LIN {X 0,Y 334.307,Z 627.426,A -85,B 0,C 180,E1 -14365.347,E2 -14365.347} C_VEL
LIN {X 0,Y 334.182,Z 628.158,A -85,B 0,C 180,E1 -14365.662,E2 -14365.662} C_VEL
LIN {X 0,Y 334.072,Z 630.189,A -85,B 0,C 180,E1 -14366.548,E2 -14366.548} C_VEL
LIN {X 0,Y 336.803,Z 644.466,A -85,B 0,C 180,E1 -14367.297,E2 -14367.297} C_VEL
LIN {X 0,Y 339.056,Z 657.276,A -85,B 0,C 180,E1 -14368.193,E2 -14368.193} C_VEL
LIN {X 0,Y 338.208,Z 670.123,A -85,B 0,C 180,E1 -14369.223,E2 -14369.223} C_VEL
LIN {X 0,Y 337.091,Z 682.489,A -85,B 0,C 180,E1 -14370.492,E2 -14370.492} C_VEL
LIN {X 0,Y 336.021,Z 693.493,A -85,B 0,C 180,E1 -14371.928,E2 -14371.928} C_VEL
LIN {X 0,Y 335.044,Z 703.461,A -85,B 0,C 180,E1 -14373.529,E2 -14373.529} C_VEL
LIN {X 0,Y 334.192,Z 711.545,A -85,B 0,C 180,E1 -14375.128,E2 -14375.128} C_VEL
LIN {X 0,Y 333.445,Z 719.422,A -85,B 0,C 180,E1 -14377.051,E2 -14377.051} C_VEL
LIN {X 0,Y 332.869,Z 725.659,A -85,B 0,C 180,E1 -14378.966,E2 -14378.966} C_VEL
LIN {X 0,Y 332.483,Z 730.459,A -85,B 0,C 180,E1 -14380.875,E2 -14380.875} C_VEL
LIN {X 0,Y 332.219,Z 734.042,A -85,B 0,C 180,E1 -14382.773,E2 -14382.773} C_VEL
LIN {X 0,Y 332.056,Z 735.815,A -85,B 0,C 180,E1 -14384.03,E2 -14384.03} C_VEL
LIN {X 0,Y 332.023,Z 737.142,A -85,B 0,C 180,E1 -14385.286,E2 -14385.286} C_VEL
LIN {X 0,Y 332.085,Z 738.091,A -85,B 0,C 180,E1 -14386.776,E2 -14386.776} C_VEL
LIN {X 0,Y 332.139,Z 738.414,A -85,B 0,C 180,E1 -14389.022,E2 -14389.022} C_VEL
LIN {X 0,Y 332.284,Z 737.954,A -85,B 0,C 180,E1 -14390.259,E2 -14390.259} C_VEL
LIN {X 0,Y 332.509,Z 737.089,A -85,B 0,C 180,E1 -14391.492,E2 -14391.492} C_VEL
LIN {X 0,Y 332.844,Z 735.56,A -85,B 0,C 180,E1 -14392.92,E2 -14392.92} C_VEL
LIN {X 0,Y 333.43,Z 731.936,A -85,B 0,C 180,E1 -14395.164,E2 -14395.164} C_VEL
LIN {X 0,Y 334.131,Z 727.836,A -85,B 0,C 180,E1 -14396.986,E2 -14396.986} C_VEL
LIN {X 0,Y 335.257,Z 721.578,A -85,B 0,C 180,E1 -14399.1,E2 -14399.1} C_VEL
LIN {X 0,Y 336.526,Z 714.727,A -85,B 0,C 180,E1 -14400.898,E2 -14400.898} C_VEL
LIN {X 0,Y 337.99,Z 706.462,A -85,B 0,C 180,E1 -14402.651,E2 -14402.651} C_VEL
LIN {X 0,Y 339.489,Z 697.76,A -85,B 0,C 180,E1 -14404.156,E2 -14404.156} C_VEL
LIN {X 0,Y 341.171,Z 687.321,A -85,B 0,C 180,E1 -14405.616,E2 -14405.616} C_VEL
LIN {X 0,Y 342.749,Z 675.77,A -85,B 0,C 180,E1 -14406.919,E2 -14406.919} C_VEL
LIN {X 0,Y 344.181,Z 663.857,A -85,B 0,C 180,E1 -14407.968,E2 -14407.968} C_VEL
LIN {X 0,Y 342.351,Z 652.946,A -85,B 0,C 180,E1 -14409.036,E2 -14409.036} C_VEL
LIN {X 0,Y 338.669,Z 640.492,A -85,B 0,C 180,E1 -14410.207,E2 -14410.207} C_VEL
LIN {X 0,Y 336.47,Z 634.41,A -85,B 0,C 180,E1 -14410.786,E2 -14410.786} C_VEL
LIN {X 0,Y 337.122,Z 626.531,A -85,B 0,C 180,E1 -14414.488,E2 -14414.488} C_VEL
LIN {X 0,Y 337.867,Z 618.773,A -85,B 0,C 180,E1 -14418.181,E2 -14418.181} C_VEL
LIN {X 0,Y 338.839,Z 611.142,A -85,B 0,C 180,E1 -14421.923,E2 -14421.923} C_VEL
LIN {X 0,Y 339.229,Z 606.089,A -85,B 0,C 180,E1 -14424.479,E2 -14424.479} C_VEL
LIN {X 0,Y 338.754,Z 601.9,A -85,B 0,C 180,E1 -14426.865,E2 -14426.865} C_VEL
LIN {X 0,Y 337.834,Z 597.015,A -85,B 0,C 180,E1 -14429.953,E2 -14429.953} C_VEL
LIN {X 0,Y 336.765,Z 592.554,A -85,B 0,C 180,E1 -14433.411,E2 -14433.411} C_VEL
LIN {X 0,Y 335.981,Z 589.986,A -85,B 0,C 180,E1 -14435.853,E2 -14435.853} C_VEL
LIN {X 0,Y 335.211,Z 587.549,A -85,B 0,C 180,E1 -14438.975,E2 -14438.975} C_VEL
LIN {X 0,Y 334.904,Z 586.539,A -85,B 0,C 180,E1 -14440.936,E2 -14440.936} C_VEL
LIN {X 0,Y 334.499,Z 586.598,A -85,B 0,C 180,E1 -14441.944,E2 -14441.944} C_VEL
LIN {X 0,Y 335.969,Z 593.434,A -85,B 0,C 180,E1 -14445.336,E2 -14445.336} C_VEL
LIN {X 0,Y 337.645,Z 601.963,A -85,B 0,C 180,E1 -14449.226,E2 -14449.226} C_VEL
LIN {X 0,Y 338.527,Z 607.233,A -85,B 0,C 180,E1 -14451.48,E2 -14451.48} C_VEL
LIN {X 0,Y 338.397,Z 611.019,A -85,B 0,C 180,E1 -14452.968,E2 -14452.968} C_VEL
LIN {X 0,Y 336.894,Z 620.66,A -85,B 0,C 180,E1 -14456.559,E2 -14456.559} C_VEL
LIN {X 0,Y 335.74,Z 629.739,A -85,B 0,C 180,E1 -14459.843,E2 -14459.843} C_VEL
LIN {X 0,Y 334.739,Z 639.124,A -85,B 0,C 180,E1 -14463.168,E2 -14463.168} C_VEL
LIN {X 0,Y 334.472,Z 641.914,A -85,B 0,C 180,E1 -14464.13,E2 -14464.13} C_VEL
LIN {X 0,Y 335.666,Z 653.856,A -85,B 0,C 180,E1 -14465.905,E2 -14465.905} C_VEL
LIN {X 0,Y 336.107,Z 656.378,A -85,B 0,C 180,E1 -14466.191,E2 -14466.191} C_VEL
LIN {X 0,Y 339.515,Z 671.747,A -85,B 0,C 180,E1 -14467.228,E2 -14467.228} C_VEL
LIN {X 0,Y 340.677,Z 682.969,A -85,B 0,C 180,E1 -14467.991,E2 -14467.991} C_VEL
LIN {X 0,Y 340.835,Z 696.04,A -85,B 0,C 180,E1 -14468.978,E2 -14468.978} C_VEL
LIN {X 0,Y 340.476,Z 708.153,A -85,B 0,C 180,E1 -14470.089,E2 -14470.089} C_VEL
LIN {X 0,Y 339.636,Z 716.55,A -85,B 0,C 180,E1 -14470.981,E2 -14470.981} C_VEL
LIN {X 0,Y 337.998,Z 727.237,A -85,B 0,C 180,E1 -14472.297,E2 -14472.297} C_VEL
LIN {X 0,Y 336.398,Z 737.43,A -85,B 0,C 180,E1 -14473.845,E2 -14473.845} C_VEL
LIN {X 0,Y 335.114,Z 745.944,A -85,B 0,C 180,E1 -14475.425,E2 -14475.425} C_VEL
LIN {X 0,Y 334.012,Z 753.925,A -85,B 0,C 180,E1 -14477.237,E2 -14477.237} C_VEL
LIN {X 0,Y 333.133,Z 760.378,A -85,B 0,C 180,E1 -14479.056,E2 -14479.056} C_VEL
LIN {X 0,Y 332.615,Z 765.591,A -85,B 0,C 180,E1 -14480.883,E2 -14480.883} C_VEL
LIN {X 0,Y 332.292,Z 769.66,A -85,B 0,C 180,E1 -14482.711,E2 -14482.711} C_VEL
LIN {X 0,Y 332.201,Z 771.787,A -85,B 0,C 180,E1 -14483.929,E2 -14483.929} C_VEL
LIN {X 0,Y 332.179,Z 773.487,A -85,B 0,C 180,E1 -14485.146,E2 -14485.146} C_VEL
LIN {X 0,Y 332.155,Z 774.712,A -85,B 0,C 180,E1 -14486.362,E2 -14486.362} C_VEL
LIN {X 0,Y 332.2,Z 775.52,A -85,B 0,C 180,E1 -14487.576,E2 -14487.576} C_VEL
LIN {X 0,Y 332.339,Z 775.927,A -85,B 0,C 180,E1 -14488.789,E2 -14488.789} C_VEL
LIN {X 0,Y 332.37,Z 775.897,A -85,B 0,C 180,E1 -14490.001,E2 -14490.001} C_VEL
LIN {X 0,Y 332.374,Z 775.4,A -85,B 0,C 180,E1 -14491.213,E2 -14491.213} C_VEL
LIN {X 0,Y 332.287,Z 774.481,A -85,B 0,C 180,E1 -14492.425,E2 -14492.425} C_VEL
LIN {X 0,Y 332.186,Z 773.133,A -85,B 0,C 180,E1 -14493.64,E2 -14493.64} C_VEL
LIN {X 0,Y 332.298,Z 771.3,A -85,B 0,C 180,E1 -14494.854,E2 -14494.854} C_VEL
LIN {X 0,Y 332.272,Z 767.789,A -85,B 0,C 180,E1 -14496.621,E2 -14496.621} C_VEL
LIN {X 0,Y 332.466,Z 762.816,A -85,B 0,C 180,E1 -14498.511,E2 -14498.511} C_VEL
LIN {X 0,Y 332.84,Z 756.668,A -85,B 0,C 180,E1 -14500.34,E2 -14500.34} C_VEL
LIN {X 0,Y 333.491,Z 748.981,A -85,B 0,C 180,E1 -14502.167,E2 -14502.167} C_VEL
LIN {X 0,Y 334.174,Z 741.078,A -85,B 0,C 180,E1 -14503.687,E2 -14503.687} C_VEL
LIN {X 0,Y 334.972,Z 732.11,A -85,B 0,C 180,E1 -14505.111,E2 -14505.111} C_VEL
LIN {X 0,Y 336.113,Z 720.935,A -85,B 0,C 180,E1 -14506.554,E2 -14506.554} C_VEL
LIN {X 0,Y 337.216,Z 709.113,A -85,B 0,C 180,E1 -14507.747,E2 -14507.747} C_VEL
LIN {X 0,Y 336.932,Z 696.74,A -85,B 0,C 180,E1 -14508.767,E2 -14508.767} C_VEL
LIN {X 0,Y 336.181,Z 683.119,A -85,B 0,C 180,E1 -14509.613,E2 -14509.613} C_VEL
LIN {X 0,Y 335.029,Z 669.463,A -85,B 0,C 180,E1 -14510.221,E2 -14510.221} C_VEL
LIN {X 0,Y 333.69,Z 657.114,A -85,B 0,C 180,E1 -14510.739,E2 -14510.739} C_VEL
LIN {X 0,Y 333.319,Z 651.132,A -85,B 0,C 180,E1 -14511.242,E2 -14511.242} C_VEL
LIN {X 0,Y 334.083,Z 638.01,A -85,B 0,C 180,E1 -14515.644,E2 -14515.644} C_VEL
LIN {X 0,Y 335.042,Z 626.598,A -85,B 0,C 180,E1 -14519.535,E2 -14519.535} C_VEL
LIN {X 0,Y 336.106,Z 615.846,A -85,B 0,C 180,E1 -14523.237,E2 -14523.237} C_VEL
LIN {X 0,Y 337.236,Z 605.77,A -85,B 0,C 180,E1 -14526.81,E2 -14526.81} C_VEL
LIN {X 0,Y 337.323,Z 602.151,A -85,B 0,C 180,E1 -14528.132,E2 -14528.132} C_VEL
LIN {X 0,Y 335.692,Z 593.071,A -85,B 0,C 180,E1 -14531.692,E2 -14531.692} C_VEL
LIN {X 0,Y 334.038,Z 584.825,A -85,B 0,C 180,E1 -14535.121,E2 -14535.121} C_VEL
LIN {X 0,Y 333.645,Z 582.926,A -85,B 0,C 180,E1 -14535.962,E2 -14535.962} C_VEL
LIN {X 0,Y 333.652,Z 582.927,A -85,B 0,C 180,E1 -14539.315,E2 -14539.315} C_VEL
LIN {X 0,Y 333.672,Z 582.919,A -85,B 0,C 180,E1 -14543.167,E2 -14543.167} C_VEL
LIN {X 0,Y 333.644,Z 582.923,A -85,B 0,C 180,E1 -14546.792,E2 -14546.792} C_VEL
LIN {X 0,Y 333.709,Z 582.914,A -85,B 0,C 180,E1 -14549.71,E2 -14549.71} C_VEL
LIN {X 0,Y 333.74,Z 582.911,A -85,B 0,C 180,E1 -14553.754,E2 -14553.754} C_VEL
LIN {X 0,Y 333.725,Z 582.914,A -85,B 0,C 180,E1 -14557.914,E2 -14557.914} C_VEL
LIN {X 0,Y 333.799,Z 582.903,A -85,B 0,C 180,E1 -14561.589,E2 -14561.589} C_VEL
LIN {X 0,Y 333.813,Z 582.901,A -85,B 0,C 180,E1 -14565.576,E2 -14565.576} C_VEL
LIN {X 0,Y 333.838,Z 582.898,A -85,B 0,C 180,E1 -14569.078,E2 -14569.078} C_VEL
LIN {X 0,Y 334.031,Z 582.876,A -85,B 0,C 180,E1 -14572.747,E2 -14572.747} C_VEL
LIN {X 0,Y 333.813,Z 582.901,A -85,B 0,C 180,E1 -14575.169,E2 -14575.169} C_VEL
LIN {X 0,Y 334.109,Z 582.864,A -85,B 0,C 180,E1 -14577.588,E2 -14577.588} C_VEL
LIN {X 0,Y 334.252,Z 582.848,A -85,B 0,C 180,E1 -14580,E2 -14580} C_VEL
LIN {X 0,Y 334.109,Z 582.869,A -85,B 0,C 180,E1 -14582.411,E2 -14582.411} C_VEL
LIN {X 0,Y 334.029,Z 582.873,A -85,B 0,C 180,E1 -14587.252,E2 -14587.252} C_VEL
LIN {X 0,Y 333.837,Z 582.899,A -85,B 0,C 180,E1 -14590.921,E2 -14590.921} C_VEL
LIN {X 0,Y 333.812,Z 582.904,A -85,B 0,C 180,E1 -14594.634,E2 -14594.634} C_VEL
LIN {X 0,Y 333.8,Z 582.906,A -85,B 0,C 180,E1 -14598.655,E2 -14598.655} C_VEL
LIN {X 0,Y 333.695,Z 582.919,A -85,B 0,C 180,E1 -14602.277,E2 -14602.277} C_VEL
LIN {X 0,Y 333.739,Z 582.913,A -85,B 0,C 180,E1 -14606.245,E2 -14606.245} C_VEL
LIN {X 0,Y 333.713,Z 582.914,A -85,B 0,C 180,E1 -14608.971,E2 -14608.971} C_VEL
LIN {X 0,Y 333.645,Z 582.926,A -85,B 0,C 180,E1 -14612.586,E2 -14612.586} C_VEL
LIN {X 0,Y 333.678,Z 582.92,A -85,B 0,C 180,E1 -14616.138,E2 -14616.138} C_VEL
LIN {X 0,Y 333.649,Z 582.921,A -85,B 0,C 180,E1 -14619.191,E2 -14619.191} C_VEL
LIN {X 0,Y 333.636,Z 582.928,A -85,B 0,C 180,E1 -14622.499,E2 -14622.499} C_VEL
LIN {X 0,Y 333.621,Z 582.925,A -85,B 0,C 180,E1 -14625.958,E2 -14625.958} C_VEL
LIN {X 0,Y 333.648,Z 582.921,A -85,B 0,C 180,E1 -14629.314,E2 -14629.314} C_VEL
LIN {X 0,Y 333.667,Z 582.919,A -85,B 0,C 180,E1 -14633.166,E2 -14633.166} C_VEL
LIN {X 0,Y 333.637,Z 582.925,A -85,B 0,C 180,E1 -14636.791,E2 -14636.791} C_VEL
LIN {X 0,Y 333.695,Z 582.915,A -85,B 0,C 180,E1 -14639.712,E2 -14639.712} C_VEL
LIN {X 0,Y 333.74,Z 582.914,A -85,B 0,C 180,E1 -14642.4,E2 -14642.4} C_VEL
LIN {X 0,Y 333.727,Z 582.912,A -85,B 0,C 180,E1 -14645.09,E2 -14645.09} C_VEL
LIN {X 0,Y 333.685,Z 582.918,A -85,B 0,C 180,E1 -14649.019,E2 -14649.019} C_VEL
LIN {X 0,Y 333.793,Z 582.903,A -85,B 0,C 180,E1 -14651.588,E2 -14651.588} C_VEL
LIN {X 0,Y 333.808,Z 582.901,A -85,B 0,C 180,E1 -14655.575,E2 -14655.575} C_VEL
LIN {X 0,Y 333.837,Z 582.899,A -85,B 0,C 180,E1 -14659.077,E2 -14659.077} C_VEL
LIN {X 0,Y 334.025,Z 582.879,A -85,B 0,C 180,E1 -14662.746,E2 -14662.746} C_VEL
LIN {X 0,Y 333.936,Z 582.889,A -85,B 0,C 180,E1 -14664.375,E2 -14664.375} C_VEL
LIN {X 0,Y 337.247,Z 594.141,A -85,B 0,C 180,E1 -14665.357,E2 -14665.357} C_VEL
LIN {X 0,Y 339.912,Z 603.552,A -85,B 0,C 180,E1 -14666.339,E2 -14666.339} C_VEL
LIN {X 0,Y 339.161,Z 614.359,A -85,B 0,C 180,E1 -14667.487,E2 -14667.487} C_VEL
LIN {X 0,Y 338.331,Z 624.38,A -85,B 0,C 180,E1 -14668.809,E2 -14668.809} C_VEL
LIN {X 0,Y 337.349,Z 634.006,A -85,B 0,C 180,E1 -14670.388,E2 -14670.388} C_VEL
LIN {X 0,Y 336.455,Z 642.391,A -85,B 0,C 180,E1 -14672.094,E2 -14672.094} C_VEL
LIN {X 0,Y 335.7,Z 649.55,A -85,B 0,C 180,E1 -14673.9,E2 -14673.9} C_VEL
LIN {X 0,Y 335.16,Z 654.395,A -85,B 0,C 180,E1 -14675.413,E2 -14675.413} C_VEL
LIN {X 0,Y 334.655,Z 659.115,A -85,B 0,C 180,E1 -14677.238,E2 -14677.238} C_VEL
LIN {X 0,Y 334.241,Z 662.263,A -85,B 0,C 180,E1 -14678.793,E2 -14678.793} C_VEL
LIN {X 0,Y 333.988,Z 665.37,A -85,B 0,C 180,E1 -14680.916,E2 -14680.916} C_VEL
LIN {X 0,Y 333.91,Z 666.609,A -85,B 0,C 180,E1 -14682.149,E2 -14682.149} C_VEL
LIN {X 0,Y 333.934,Z 667.776,A -85,B 0,C 180,E1 -14684.509,E2 -14684.509} C_VEL
LIN {X 0,Y 334.096,Z 667.803,A -85,B 0,C 180,E1 -14685.869,E2 -14685.869} C_VEL
LIN {X 0,Y 334.249,Z 667.398,A -85,B 0,C 180,E1 -14687.118,E2 -14687.118} C_VEL
LIN {X 0,Y 334.756,Z 665.826,A -85,B 0,C 180,E1 -14689.137,E2 -14689.137} C_VEL
LIN {X 0,Y 335.561,Z 662.549,A -85,B 0,C 180,E1 -14691.5,E2 -14691.5} C_VEL
LIN {X 0,Y 336.414,Z 658.718,A -85,B 0,C 180,E1 -14693.385,E2 -14693.385} C_VEL
LIN {X 0,Y 337.428,Z 653.667,A -85,B 0,C 180,E1 -14695.274,E2 -14695.274} C_VEL
LIN {X 0,Y 338.646,Z 647.151,A -85,B 0,C 180,E1 -14697.165,E2 -14697.165} C_VEL
LIN {X 0,Y 340.117,Z 638.895,A -85,B 0,C 180,E1 -14699.05,E2 -14699.05} C_VEL
LIN {X 0,Y 341.533,Z 630.236,A -85,B 0,C 180,E1 -14700.633,E2 -14700.633} C_VEL
LIN {X 0,Y 342.769,Z 620.752,A -85,B 0,C 180,E1 -14702.04,E2 -14702.04} C_VEL
LIN {X 0,Y 343.821,Z 612.329,A -85,B 0,C 180,E1 -14703.064,E2 -14703.064} C_VEL
LIN {X 0,Y 343.026,Z 608.47,A -85,B 0,C 180,E1 -14703.584,E2 -14703.584} C_VEL
LIN {X 0,Y 339.681,Z 597.97,A -85,B 0,C 180,E1 -14704.932,E2 -14704.932} C_VEL
LIN {X 0,Y 335.979,Z 588.61,A -85,B 0,C 180,E1 -14706.014,E2 -14706.014} C_VEL
LIN {X 0,Y 334.161,Z 585.204,A -85,B 0,C 180,E1 -14706.423,E2 -14706.423} C_VEL
LIN {X 0,Y 335.344,Z 592.252,A -85,B 0,C 180,E1 -14709.73,E2 -14709.73} C_VEL
LIN {X 0,Y 335.556,Z 597.441,A -85,B 0,C 180,E1 -14712.082,E2 -14712.082} C_VEL
LIN {X 0,Y 335.238,Z 605.006,A -85,B 0,C 180,E1 -14715.46,E2 -14715.46} C_VEL
LIN {X 0,Y 334.771,Z 613.229,A -85,B 0,C 180,E1 -14719.09,E2 -14719.09} C_VEL
LIN {X 0,Y 334.502,Z 620.877,A -85,B 0,C 180,E1 -14722.462,E2 -14722.462} C_VEL
LIN {X 0,Y 334.182,Z 628.158,A -85,B 0,C 180,E1 -14725.662,E2 -14725.662} C_VEL
LIN {X 0,Y 334.028,Z 630.109,A -85,B 0,C 180,E1 -14726.142,E2 -14726.142} C_VEL
LIN {X 0,Y 333.66,Z 633.986,A -85,B 0,C 180,E1 -14726.58,E2 -14726.58} C_VEL
LIN {X 0,Y 333.01,Z 640.169,A -85,B 0,C 180,E1 -14726.906,E2 -14726.906} C_VEL
LIN {X 0,Y 331.643,Z 652.47,A -85,B 0,C 180,E1 -14727.534,E2 -14727.534} C_VEL
LIN {X 0,Y 331.953,Z 656.912,A -85,B 0,C 180,E1 -14727.855,E2 -14727.855} C_VEL
LIN {X 0,Y 331.934,Z 661.668,A -85,B 0,C 180,E1 -14728.218,E2 -14728.218} C_VEL
LIN {X 0,Y 331.085,Z 672.909,A -85,B 0,C 180,E1 -14729.196,E2 -14729.196} C_VEL
LIN {X 0,Y 329.945,Z 684.661,A -85,B 0,C 180,E1 -14730.491,E2 -14730.491} C_VEL
LIN {X 0,Y 328.887,Z 695.368,A -85,B 0,C 180,E1 -14731.959,E2 -14731.959} C_VEL
LIN {X 0,Y 327.925,Z 704.858,A -85,B 0,C 180,E1 -14733.568,E2 -14733.568} C_VEL
LIN {X 0,Y 326.893,Z 714.317,A -85,B 0,C 180,E1 -14735.553,E2 -14735.553} C_VEL
LIN {X 0,Y 326.186,Z 722.052,A -85,B 0,C 180,E1 -14737.63,E2 -14737.63} C_VEL
LIN {X 0,Y 325.593,Z 728.357,A -85,B 0,C 180,E1 -14739.797,E2 -14739.797} C_VEL
LIN {X 0,Y 325.274,Z 732.938,A -85,B 0,C 180,E1 -14741.925,E2 -14741.925} C_VEL
LIN {X 0,Y 325.009,Z 735.702,A -85,B 0,C 180,E1 -14743.674,E2 -14743.674} C_VEL
LIN {X 0,Y 324.943,Z 737.164,A -85,B 0,C 180,E1 -14744.958,E2 -14744.958} C_VEL
LIN {X 0,Y 324.993,Z 738.421,A -85,B 0,C 180,E1 -14746.68,E2 -14746.68} C_VEL
LIN {X 0,Y 325.05,Z 738.884,A -85,B 0,C 180,E1 -14748.78,E2 -14748.78} C_VEL
LIN {X 0,Y 325.179,Z 738.61,A -85,B 0,C 180,E1 -14750.044,E2 -14750.044} C_VEL
LIN {X 0,Y 325.389,Z 737.888,A -85,B 0,C 180,E1 -14751.305,E2 -14751.305} C_VEL
LIN {X 0,Y 325.784,Z 736.389,A -85,B 0,C 180,E1 -14752.89,E2 -14752.89} C_VEL
LIN {X 0,Y 326.358,Z 733.212,A -85,B 0,C 180,E1 -14755.059,E2 -14755.059} C_VEL
LIN {X 0,Y 327.053,Z 729.361,A -85,B 0,C 180,E1 -14756.921,E2 -14756.921} C_VEL
LIN {X 0,Y 328.051,Z 724.353,A -85,B 0,C 180,E1 -14758.773,E2 -14758.773} C_VEL
LIN {X 0,Y 329.521,Z 716.955,A -85,B 0,C 180,E1 -14760.917,E2 -14760.917} C_VEL
LIN {X 0,Y 331.111,Z 708.756,A -85,B 0,C 180,E1 -14762.778,E2 -14762.778} C_VEL
LIN {X 0,Y 332.902,Z 699.065,A -85,B 0,C 180,E1 -14764.541,E2 -14764.541} C_VEL
LIN {X 0,Y 334.651,Z 688.804,A -85,B 0,C 180,E1 -14766.028,E2 -14766.028} C_VEL
LIN {X 0,Y 336.327,Z 677.58,A -85,B 0,C 180,E1 -14767.354,E2 -14767.354} C_VEL
LIN {X 0,Y 337.802,Z 666.688,A -85,B 0,C 180,E1 -14768.375,E2 -14768.375} C_VEL
LIN {X 0,Y 337.714,Z 663.23,A -85,B 0,C 180,E1 -14768.709,E2 -14768.709} C_VEL
LIN {X 0,Y 336.082,Z 654.225,A -85,B 0,C 180,E1 -14769.631,E2 -14769.631} C_VEL
LIN {X 0,Y 332.251,Z 641.507,A -85,B 0,C 180,E1 -14770.925,E2 -14770.925} C_VEL
LIN {X 0,Y 329.847,Z 634.887,A -85,B 0,C 180,E1 -14771.616,E2 -14771.616} C_VEL
LIN {X 0,Y 330.567,Z 627.015,A -85,B 0,C 180,E1 -14775.412,E2 -14775.412} C_VEL
LIN {X 0,Y 331.423,Z 619.333,A -85,B 0,C 180,E1 -14779.189,E2 -14779.189} C_VEL
LIN {X 0,Y 332.525,Z 611.787,A -85,B 0,C 180,E1 -14783.017,E2 -14783.017} C_VEL
LIN {X 0,Y 332.695,Z 608.178,A -85,B 0,C 180,E1 -14784.992,E2 -14784.992} C_VEL
LIN {X 0,Y 332.133,Z 603.529,A -85,B 0,C 180,E1 -14787.745,E2 -14787.745} C_VEL
LIN {X 0,Y 331.628,Z 600.722,A -85,B 0,C 180,E1 -14789.673,E2 -14789.673} C_VEL
LIN {X 0,Y 331.003,Z 597.785,A -85,B 0,C 180,E1 -14792.061,E2 -14792.061} C_VEL
LIN {X 0,Y 330.159,Z 594.47,A -85,B 0,C 180,E1 -14795.082,E2 -14795.082} C_VEL
LIN {X 0,Y 329.451,Z 592.024,A -85,B 0,C 180,E1 -14798.218,E2 -14798.218} C_VEL
LIN {X 0,Y 329.268,Z 591.122,A -85,B 0,C 180,E1 -14799.817,E2 -14799.817} C_VEL
LIN {X 0,Y 328.816,Z 590.694,A -85,B 0,C 180,E1 -14801.578,E2 -14801.578} C_VEL
LIN {X 0,Y 328.227,Z 590.987,A -85,B 0,C 180,E1 -14803.171,E2 -14803.171} C_VEL
LIN {X 0,Y 329.616,Z 597.705,A -85,B 0,C 180,E1 -14806.465,E2 -14806.465} C_VEL
LIN {X 0,Y 331.329,Z 606.54,A -85,B 0,C 180,E1 -14810.482,E2 -14810.482} C_VEL
LIN {X 0,Y 331.645,Z 610.34,A -85,B 0,C 180,E1 -14812.083,E2 -14812.083} C_VEL
LIN {X 0,Y 330.527,Z 617.8,A -85,B 0,C 180,E1 -14814.965,E2 -14814.965} C_VEL
LIN {X 0,Y 328.965,Z 628.992,A -85,B 0,C 180,E1 -14819.155,E2 -14819.155} C_VEL
LIN {X 0,Y 327.834,Z 638.822,A -85,B 0,C 180,E1 -14822.685,E2 -14822.685} C_VEL
LIN {X 0,Y 329.077,Z 652.142,A -85,B 0,C 180,E1 -14824.885,E2 -14824.885} C_VEL
LIN {X 0,Y 329.478,Z 655.573,A -85,B 0,C 180,E1 -14825.358,E2 -14825.358} C_VEL
LIN {X 0,Y 332.741,Z 669.626,A -85,B 0,C 180,E1 -14826.398,E2 -14826.398} C_VEL
LIN {X 0,Y 334.185,Z 679.781,A -85,B 0,C 180,E1 -14827.127,E2 -14827.127} C_VEL
LIN {X 0,Y 334.605,Z 692.047,A -85,B 0,C 180,E1 -14828.062,E2 -14828.062} C_VEL
LIN {X 0,Y 334.086,Z 704.814,A -85,B 0,C 180,E1 -14829.209,E2 -14829.209} C_VEL
LIN {X 0,Y 333.568,Z 713.591,A -85,B 0,C 180,E1 -14830.14,E2 -14830.14} C_VEL
LIN {X 0,Y 331.673,Z 725.803,A -85,B 0,C 180,E1 -14831.629,E2 -14831.629} C_VEL
LIN {X 0,Y 330.111,Z 734.831,A -85,B 0,C 180,E1 -14832.98,E2 -14832.98} C_VEL
LIN {X 0,Y 328.566,Z 743.813,A -85,B 0,C 180,E1 -14834.622,E2 -14834.622} C_VEL
LIN {X 0,Y 327.302,Z 752.817,A -85,B 0,C 180,E1 -14836.655,E2 -14836.655} C_VEL
LIN {X 0,Y 326.347,Z 758.397,A -85,B 0,C 180,E1 -14838.196,E2 -14838.196} C_VEL
LIN {X 0,Y 325.739,Z 763.915,A -85,B 0,C 180,E1 -14840.062,E2 -14840.062} C_VEL
LIN {X 0,Y 325.33,Z 768.255,A -85,B 0,C 180,E1 -14841.929,E2 -14841.929} C_VEL
LIN {X 0,Y 325.1,Z 771.779,A -85,B 0,C 180,E1 -14843.952,E2 -14843.952} C_VEL
LIN {X 0,Y 325.077,Z 774.363,A -85,B 0,C 180,E1 -14846.282,E2 -14846.282} C_VEL
LIN {X 0,Y 325.102,Z 775.141,A -85,B 0,C 180,E1 -14847.523,E2 -14847.523} C_VEL
LIN {X 0,Y 325.256,Z 775.515,A -85,B 0,C 180,E1 -14848.763,E2 -14848.763} C_VEL
LIN {X 0,Y 325.307,Z 775.416,A -85,B 0,C 180,E1 -14850.001,E2 -14850.001} C_VEL
LIN {X 0,Y 325.31,Z 774.887,A -85,B 0,C 180,E1 -14851.239,E2 -14851.239} C_VEL
LIN {X 0,Y 325.193,Z 773.936,A -85,B 0,C 180,E1 -14852.478,E2 -14852.478} C_VEL
LIN {X 0,Y 325.112,Z 772.531,A -85,B 0,C 180,E1 -14853.719,E2 -14853.719} C_VEL
LIN {X 0,Y 325.132,Z 769.332,A -85,B 0,C 180,E1 -14855.694,E2 -14855.694} C_VEL
LIN {X 0,Y 325.273,Z 765.453,A -85,B 0,C 180,E1 -14857.45,E2 -14857.45} C_VEL
LIN {X 0,Y 325.57,Z 759.097,A -85,B 0,C 180,E1 -14859.632,E2 -14859.632} C_VEL
LIN {X 0,Y 326.085,Z 752.116,A -85,B 0,C 180,E1 -14861.501,E2 -14861.501} C_VEL
LIN {X 0,Y 326.85,Z 743.332,A -85,B 0,C 180,E1 -14863.366,E2 -14863.366} C_VEL
LIN {X 0,Y 327.64,Z 736.308,A -85,B 0,C 180,E1 -14864.599,E2 -14864.599} C_VEL
LIN {X 0,Y 328.359,Z 727.944,A -85,B 0,C 180,E1 -14865.846,E2 -14865.846} C_VEL
LIN {X 0,Y 329.501,Z 716.695,A -85,B 0,C 180,E1 -14867.215,E2 -14867.215} C_VEL
LIN {X 0,Y 330.29,Z 707.365,A -85,B 0,C 180,E1 -14868.132,E2 -14868.132} C_VEL
LIN {X 0,Y 329.856,Z 694.398,A -85,B 0,C 180,E1 -14869.188,E2 -14869.188} C_VEL
LIN {X 0,Y 329.033,Z 680.338,A -85,B 0,C 180,E1 -14870.051,E2 -14870.051} C_VEL
LIN {X 0,Y 326.686,Z 656.328,A -85,B 0,C 180,E1 -14871.122,E2 -14871.122} C_VEL
LIN {X 0,Y 326.275,Z 649.984,A -85,B 0,C 180,E1 -14871.692,E2 -14871.692} C_VEL
LIN {X 0,Y 327.082,Z 637.084,A -85,B 0,C 180,E1 -14876.135,E2 -14876.135} C_VEL
LIN {X 0,Y 327.972,Z 627.324,A -85,B 0,C 180,E1 -14879.53,E2 -14879.53} C_VEL
LIN {X 0,Y 328.951,Z 617.603,A -85,B 0,C 180,E1 -14882.966,E2 -14882.966} C_VEL
LIN {X 0,Y 330.128,Z 607.576,A -85,B 0,C 180,E1 -14886.591,E2 -14886.591} C_VEL
LIN {X 0,Y 330.372,Z 603.542,A -85,B 0,C 180,E1 -14888.092,E2 -14888.092} C_VEL
LIN {X 0,Y 328.799,Z 594.835,A -85,B 0,C 180,E1 -14891.572,E2 -14891.572} C_VEL
LIN {X 0,Y 327.118,Z 586.394,A -85,B 0,C 180,E1 -14895.154,E2 -14895.154} C_VEL
LIN {X 0,Y 326.594,Z 583.805,A -85,B 0,C 180,E1 -14896.373,E2 -14896.373} C_VEL
LIN {X 0,Y 326.597,Z 583.804,A -85,B 0,C 180,E1 -14899.791,E2 -14899.791} C_VEL
LIN {X 0,Y 326.637,Z 583.796,A -85,B 0,C 180,E1 -14902.954,E2 -14902.954} C_VEL
LIN {X 0,Y 326.613,Z 583.801,A -85,B 0,C 180,E1 -14905.981,E2 -14905.981} C_VEL
LIN {X 0,Y 326.666,Z 583.797,A -85,B 0,C 180,E1 -14910.341,E2 -14910.341} C_VEL
LIN {X 0,Y 326.695,Z 583.791,A -85,B 0,C 180,E1 -14914.516,E2 -14914.516} C_VEL
LIN {X 0,Y 326.651,Z 583.797,A -85,B 0,C 180,E1 -14918.545,E2 -14918.545} C_VEL
LIN {X 0,Y 326.75,Z 583.781,A -85,B 0,C 180,E1 -14921.177,E2 -14921.177} C_VEL
LIN {X 0,Y 326.768,Z 583.778,A -85,B 0,C 180,E1 -14925.433,E2 -14925.433} C_VEL
LIN {X 0,Y 326.775,Z 583.779,A -85,B 0,C 180,E1 -14928.839,E2 -14928.839} C_VEL
LIN {X 0,Y 326.982,Z 583.755,A -85,B 0,C 180,E1 -14932.59,E2 -14932.59} C_VEL
LIN {X 0,Y 326.78,Z 583.777,A -85,B 0,C 180,E1 -14935.064,E2 -14935.064} C_VEL
LIN {X 0,Y 327.05,Z 583.743,A -85,B 0,C 180,E1 -14937.536,E2 -14937.536} C_VEL
LIN {X 0,Y 327.203,Z 583.726,A -85,B 0,C 180,E1 -14940,E2 -14940} C_VEL
LIN {X 0,Y 327.049,Z 583.747,A -85,B 0,C 180,E1 -14942.463,E2 -14942.463} C_VEL
LIN {X 0,Y 326.975,Z 583.751,A -85,B 0,C 180,E1 -14946.66,E2 -14946.66} C_VEL
LIN {X 0,Y 326.818,Z 583.773,A -85,B 0,C 180,E1 -14949.906,E2 -14949.906} C_VEL
LIN {X 0,Y 326.763,Z 583.779,A -85,B 0,C 180,E1 -14953.685,E2 -14953.685} C_VEL
LIN {X 0,Y 326.702,Z 583.785,A -85,B 0,C 180,E1 -14957.527,E2 -14957.527} C_VEL
LIN {X 0,Y 326.668,Z 583.793,A -85,B 0,C 180,E1 -14960.134,E2 -14960.134} C_VEL
LIN {X 0,Y 326.655,Z 583.795,A -85,B 0,C 180,E1 -14964.128,E2 -14964.128} C_VEL
LIN {X 0,Y 326.688,Z 583.789,A -85,B 0,C 180,E1 -14966.857,E2 -14966.857} C_VEL
LIN {X 0,Y 326.641,Z 583.798,A -85,B 0,C 180,E1 -14970.61,E2 -14970.61} C_VEL
LIN {X 0,Y 326.609,Z 583.799,A -85,B 0,C 180,E1 -14974.019,E2 -14974.019} C_VEL
LIN {X 0,Y 326.63,Z 583.795,A -85,B 0,C 180,E1 -14977.238,E2 -14977.238} C_VEL
LIN {X 0,Y 326.579,Z 583.802,A -85,B 0,C 180,E1 -14981.13,E2 -14981.13} C_VEL
LIN {X 0,Y 326.558,Z 583.807,A -85,B 0,C 180,E1 -14984.747,E2 -14984.747} C_VEL
LIN {X 0,Y 326.577,Z 583.804,A -85,B 0,C 180,E1 -14988.153,E2 -14988.153} C_VEL
LIN {X 0,Y 326.625,Z 583.795,A -85,B 0,C 180,E1 -14991.391,E2 -14991.391} C_VEL
LIN {X 0,Y 326.621,Z 583.799,A -85,B 0,C 180,E1 -14994.85,E2 -14994.85} C_VEL
LIN {X 0,Y 326.608,Z 583.798,A -85,B 0,C 180,E1 -14997.455,E2 -14997.455} C_VEL
LIN {X 0,Y 326.648,Z 583.797,A -85,B 0,C 180,E1 -15000.339,E2 -15000.339} C_VEL
LIN {X 0,Y 326.69,Z 583.793,A -85,B 0,C 180,E1 -15004.515,E2 -15004.515} C_VEL
LIN {X 0,Y 326.648,Z 583.799,A -85,B 0,C 180,E1 -15008.544,E2 -15008.544} C_VEL
LIN {X 0,Y 326.744,Z 583.782,A -85,B 0,C 180,E1 -15011.176,E2 -15011.176} C_VEL
LIN {X 0,Y 326.762,Z 583.779,A -85,B 0,C 180,E1 -15015.432,E2 -15015.432} C_VEL
LIN {X 0,Y 326.773,Z 583.781,A -85,B 0,C 180,E1 -15018.838,E2 -15018.838} C_VEL
LIN {X 0,Y 326.979,Z 583.758,A -85,B 0,C 180,E1 -15022.589,E2 -15022.589} C_VEL
LIN {X 0,Y 326.967,Z 583.755,A -85,B 0,C 180,E1 -15024.023,E2 -15024.023} C_VEL
LIN {X 0,Y 330.506,Z 596.027,A -85,B 0,C 180,E1 -15025.12,E2 -15025.12} C_VEL
LIN {X 0,Y 332.996,Z 604.816,A -85,B 0,C 180,E1 -15026.068,E2 -15026.068} C_VEL
LIN {X 0,Y 332.268,Z 615.812,A -85,B 0,C 180,E1 -15027.271,E2 -15027.271} C_VEL
LIN {X 0,Y 331.505,Z 624.783,A -85,B 0,C 180,E1 -15028.48,E2 -15028.48} C_VEL
LIN {X 0,Y 330.55,Z 634.055,A -85,B 0,C 180,E1 -15029.999,E2 -15029.999} C_VEL
LIN {X 0,Y 329.542,Z 643.014,A -85,B 0,C 180,E1 -15031.832,E2 -15031.832} C_VEL
LIN {X 0,Y 328.756,Z 650.239,A -85,B 0,C 180,E1 -15033.676,E2 -15033.676} C_VEL
LIN {X 0,Y 328.084,Z 656.049,A -85,B 0,C 180,E1 -15035.53,E2 -15035.53} C_VEL
LIN {X 0,Y 327.591,Z 660.63,A -85,B 0,C 180,E1 -15037.395,E2 -15037.395} C_VEL
LIN {X 0,Y 327.204,Z 663.474,A -85,B 0,C 180,E1 -15038.877,E2 -15038.877} C_VEL
LIN {X 0,Y 326.937,Z 666.651,A -85,B 0,C 180,E1 -15041.154,E2 -15041.154} C_VEL
LIN {X 0,Y 326.888,Z 667.78,A -85,B 0,C 180,E1 -15042.414,E2 -15042.414} C_VEL
LIN {X 0,Y 326.981,Z 668.849,A -85,B 0,C 180,E1 -15044.946,E2 -15044.946} C_VEL
LIN {X 0,Y 327.126,Z 668.787,A -85,B 0,C 180,E1 -15046.217,E2 -15046.217} C_VEL
LIN {X 0,Y 327.307,Z 668.284,A -85,B 0,C 180,E1 -15047.493,E2 -15047.493} C_VEL
LIN {X 0,Y 327.81,Z 666.786,A -85,B 0,C 180,E1 -15049.383,E2 -15049.383} C_VEL
LIN {X 0,Y 328.752,Z 663.195,A -85,B 0,C 180,E1 -15051.968,E2 -15051.968} C_VEL
LIN {X 0,Y 329.686,Z 659.224,A -85,B 0,C 180,E1 -15053.891,E2 -15053.891} C_VEL
LIN {X 0,Y 331.005,Z 652.971,A -85,B 0,C 180,E1 -15056.139,E2 -15056.139} C_VEL
LIN {X 0,Y 332.364,Z 646.047,A -85,B 0,C 180,E1 -15058.064,E2 -15058.064} C_VEL
LIN {X 0,Y 333.698,Z 638.851,A -85,B 0,C 180,E1 -15059.664,E2 -15059.664} C_VEL
LIN {X 0,Y 335.274,Z 629.072,A -85,B 0,C 180,E1 -15061.409,E2 -15061.409} C_VEL
LIN {X 0,Y 336.671,Z 618.874,A -85,B 0,C 180,E1 -15062.869,E2 -15062.869} C_VEL
LIN {X 0,Y 337.267,Z 613.36,A -85,B 0,C 180,E1 -15063.539,E2 -15063.539} C_VEL
LIN {X 0,Y 334.295,Z 603.421,A -85,B 0,C 180,E1 -15064.925,E2 -15064.925} C_VEL
LIN {X 0,Y 330.701,Z 593.702,A -85,B 0,C 180,E1 -15066.142,E2 -15066.142} C_VEL
LIN {X 0,Y 328.887,Z 590.413,A -85,B 0,C 180,E1 -15066.576,E2 -15066.576} C_VEL
LIN {X 0,Y 327.449,Z 588.013,A -85,B 0,C 180,E1 -15066.884,E2 -15066.884} C_VEL
LIN {X 0,Y 327.398,Z 587.848,A -85,B 0,C 180,E1 -15066.944,E2 -15066.944} C_VEL
LIN {X 0,Y 328.439,Z 594.121,A -85,B 0,C 180,E1 -15069.935,E2 -15069.935} C_VEL
LIN {X 0,Y 328.549,Z 599.435,A -85,B 0,C 180,E1 -15072.359,E2 -15072.359} C_VEL
LIN {X 0,Y 328.187,Z 607.303,A -85,B 0,C 180,E1 -15075.896,E2 -15075.896} C_VEL
LIN {X 0,Y 327.707,Z 616.378,A -85,B 0,C 180,E1 -15079.956,E2 -15079.956} C_VEL
LIN {X 0,Y 327.334,Z 625.058,A -85,B 0,C 180,E1 -15083.813,E2 -15083.813} C_VEL
LIN {X 0,Y 327.107,Z 630.627,A -85,B 0,C 180,E1 -15086.246,E2 -15086.246} C_VEL
LIN {X 0,Y 329.67,Z 644.256,A -85,B 0,C 180,E1 -15086.961,E2 -15086.961} C_VEL
LIN {X 0,Y 331.953,Z 656.912,A -85,B 0,C 180,E1 -15087.855,E2 -15087.855} C_VEL
LIN {X 0,Y 332.055,Z 660.475,A -85,B 0,C 180,E1 -15088.123,E2 -15088.123} C_VEL
LIN {X 0,Y 331.332,Z 664.021,A -85,B 0,C 180,E1 -15088.379,E2 -15088.379} C_VEL
LIN {X 0,Y 328.442,Z 670.852,A -85,B 0,C 180,E1 -15088.88,E2 -15088.88} C_VEL
LIN {X 0,Y 324.347,Z 679.17,A -85,B 0,C 180,E1 -15089.608,E2 -15089.608} C_VEL
LIN {X 0,Y 323.067,Z 684.138,A -85,B 0,C 180,E1 -15090.166,E2 -15090.166} C_VEL
LIN {X 0,Y 321.977,Z 694.946,A -85,B 0,C 180,E1 -15091.657,E2 -15091.657} C_VEL
LIN {X 0,Y 320.934,Z 704.758,A -85,B 0,C 180,E1 -15093.326,E2 -15093.326} C_VEL
LIN {X 0,Y 319.898,Z 714.196,A -85,B 0,C 180,E1 -15095.329,E2 -15095.329} C_VEL
LIN {X 0,Y 319.212,Z 721.397,A -85,B 0,C 180,E1 -15097.243,E2 -15097.243} C_VEL
LIN {X 0,Y 318.587,Z 727.599,A -85,B 0,C 180,E1 -15099.332,E2 -15099.332} C_VEL
LIN {X 0,Y 318.256,Z 732.084,A -85,B 0,C 180,E1 -15101.282,E2 -15101.282} C_VEL
LIN {X 0,Y 317.958,Z 735.534,A -85,B 0,C 180,E1 -15103.301,E2 -15103.301} C_VEL
LIN {X 0,Y 317.856,Z 737.166,A -85,B 0,C 180,E1 -15104.614,E2 -15104.614} C_VEL
LIN {X 0,Y 317.902,Z 738.748,A -85,B 0,C 180,E1 -15106.581,E2 -15106.581} C_VEL
LIN {X 0,Y 317.972,Z 739.347,A -85,B 0,C 180,E1 -15108.527,E2 -15108.527} C_VEL
LIN {X 0,Y 318.07,Z 739.194,A -85,B 0,C 180,E1 -15109.819,E2 -15109.819} C_VEL
LIN {X 0,Y 318.269,Z 738.641,A -85,B 0,C 180,E1 -15111.108,E2 -15111.108} C_VEL
LIN {X 0,Y 318.707,Z 737.16,A -85,B 0,C 180,E1 -15112.883,E2 -15112.883} C_VEL
LIN {X 0,Y 319.264,Z 734.414,A -85,B 0,C 180,E1 -15114.949,E2 -15114.949} C_VEL
LIN {X 0,Y 319.979,Z 730.824,A -85,B 0,C 180,E1 -15116.853,E2 -15116.853} C_VEL
LIN {X 0,Y 321.029,Z 726.139,A -85,B 0,C 180,E1 -15118.746,E2 -15118.746} C_VEL
LIN {X 0,Y 322.503,Z 719.113,A -85,B 0,C 180,E1 -15120.937,E2 -15120.937} C_VEL
LIN {X 0,Y 324.163,Z 711.336,A -85,B 0,C 180,E1 -15122.837,E2 -15122.837} C_VEL
LIN {X 0,Y 325.613,Z 703.874,A -85,B 0,C 180,E1 -15124.333,E2 -15124.333} C_VEL
LIN {X 0,Y 327.566,Z 693.65,A -85,B 0,C 180,E1 -15126.004,E2 -15126.004} C_VEL
LIN {X 0,Y 329.574,Z 682.145,A -85,B 0,C 180,E1 -15127.505,E2 -15127.505} C_VEL
LIN {X 0,Y 331.209,Z 670.847,A -85,B 0,C 180,E1 -15128.673,E2 -15128.673} C_VEL
LIN {X 0,Y 331.698,Z 666.656,A -85,B 0,C 180,E1 -15129.05,E2 -15129.05} C_VEL
LIN {X 0,Y 330.011,Z 656.334,A -85,B 0,C 180,E1 -15130.185,E2 -15130.185} C_VEL
LIN {X 0,Y 326.514,Z 644.362,A -85,B 0,C 180,E1 -15131.49,E2 -15131.49} C_VEL
LIN {X 0,Y 323.242,Z 635.605,A -85,B 0,C 180,E1 -15132.437,E2 -15132.437} C_VEL
LIN {X 0,Y 324.076,Z 627.665,A -85,B 0,C 180,E1 -15136.375,E2 -15136.375} C_VEL
LIN {X 0,Y 325.104,Z 620,A -85,B 0,C 180,E1 -15140.236,E2 -15140.236} C_VEL
LIN {X 0,Y 326.038,Z 613.768,A -85,B 0,C 180,E1 -15143.503,E2 -15143.503} C_VEL
LIN {X 0,Y 326.191,Z 610.316,A -85,B 0,C 180,E1 -15145.526,E2 -15145.526} C_VEL
LIN {X 0,Y 325.647,Z 605.906,A -85,B 0,C 180,E1 -15148.347,E2 -15148.347} C_VEL
LIN {X 0,Y 325.326,Z 603.606,A -85,B 0,C 180,E1 -15150.221,E2 -15150.221} C_VEL
LIN {X 0,Y 324.665,Z 600.56,A -85,B 0,C 180,E1 -15152.764,E2 -15152.764} C_VEL
LIN {X 0,Y 324.021,Z 597.646,A -85,B 0,C 180,E1 -15155.848,E2 -15155.848} C_VEL
LIN {X 0,Y 323.492,Z 595.59,A -85,B 0,C 180,E1 -15159.053,E2 -15159.053} C_VEL
LIN {X 0,Y 323.251,Z 595.032,A -85,B 0,C 180,E1 -15160.712,E2 -15160.712} C_VEL
LIN {X 0,Y 322.691,Z 595.123,A -85,B 0,C 180,E1 -15162.467,E2 -15162.467} C_VEL
LIN {X 0,Y 322.06,Z 596.005,A -85,B 0,C 180,E1 -15164.73,E2 -15164.73} C_VEL
LIN {X 0,Y 323.215,Z 602.073,A -85,B 0,C 180,E1 -15167.672,E2 -15167.672} C_VEL
LIN {X 0,Y 324.345,Z 607.709,A -85,B 0,C 180,E1 -15170.269,E2 -15170.269} C_VEL
LIN {X 0,Y 324.696,Z 611.622,A -85,B 0,C 180,E1 -15171.959,E2 -15171.959} C_VEL
LIN {X 0,Y 323.547,Z 618.943,A -85,B 0,C 180,E1 -15174.858,E2 -15174.858} C_VEL
LIN {X 0,Y 322.169,Z 628.251,A -85,B 0,C 180,E1 -15178.431,E2 -15178.431} C_VEL
LIN {X 0,Y 321.31,Z 634.751,A -85,B 0,C 180,E1 -15180.846,E2 -15180.846} C_VEL
LIN {X 0,Y 322.119,Z 646.127,A -85,B 0,C 180,E1 -15183.038,E2 -15183.038} C_VEL
LIN {X 0,Y 322.988,Z 654.983,A -85,B 0,C 180,E1 -15184.49,E2 -15184.49} C_VEL
LIN {X 0,Y 326.338,Z 668.908,A -85,B 0,C 180,E1 -15185.596,E2 -15185.596} C_VEL
LIN {X 0,Y 327.957,Z 679.637,A -85,B 0,C 180,E1 -15186.435,E2 -15186.435} C_VEL
LIN {X 0,Y 328.319,Z 692.633,A -85,B 0,C 180,E1 -15187.479,E2 -15187.479} C_VEL
LIN {X 0,Y 327.642,Z 706.437,A -85,B 0,C 180,E1 -15188.78,E2 -15188.78} C_VEL
LIN {X 0,Y 326.993,Z 714.757,A -85,B 0,C 180,E1 -15189.724,E2 -15189.724} C_VEL
LIN {X 0,Y 325.001,Z 726.544,A -85,B 0,C 180,E1 -15191.238,E2 -15191.238} C_VEL
LIN {X 0,Y 323.347,Z 735.355,A -85,B 0,C 180,E1 -15192.612,E2 -15192.612} C_VEL
LIN {X 0,Y 321.556,Z 745.472,A -85,B 0,C 180,E1 -15194.561,E2 -15194.561} C_VEL
LIN {X 0,Y 320.382,Z 752.977,A -85,B 0,C 180,E1 -15196.362,E2 -15196.362} C_VEL
LIN {X 0,Y 319.1,Z 760.358,A -85,B 0,C 180,E1 -15198.568,E2 -15198.568} C_VEL
LIN {X 0,Y 318.535,Z 765.377,A -85,B 0,C 180,E1 -15200.476,E2 -15200.476} C_VEL
LIN {X 0,Y 318.17,Z 769.269,A -85,B 0,C 180,E1 -15202.385,E2 -15202.385} C_VEL
LIN {X 0,Y 318.024,Z 771.716,A -85,B 0,C 180,E1 -15203.967,E2 -15203.967} C_VEL
LIN {X 0,Y 318,Z 774.021,A -85,B 0,C 180,E1 -15206.2,E2 -15206.2} C_VEL
LIN {X 0,Y 318.009,Z 774.764,A -85,B 0,C 180,E1 -15207.468,E2 -15207.468} C_VEL
LIN {X 0,Y 318.174,Z 775.081,A -85,B 0,C 180,E1 -15208.735,E2 -15208.735} C_VEL
LIN {X 0,Y 318.245,Z 774.935,A -85,B 0,C 180,E1 -15210.001,E2 -15210.001} C_VEL
LIN {X 0,Y 318.246,Z 774.372,A -85,B 0,C 180,E1 -15211.267,E2 -15211.267} C_VEL
LIN {X 0,Y 318.1,Z 773.378,A -85,B 0,C 180,E1 -15212.534,E2 -15212.534} C_VEL
LIN {X 0,Y 318.04,Z 771.9,A -85,B 0,C 180,E1 -15213.802,E2 -15213.802} C_VEL
LIN {X 0,Y 318.048,Z 768.948,A -85,B 0,C 180,E1 -15215.651,E2 -15215.651} C_VEL
LIN {X 0,Y 318.203,Z 764.647,A -85,B 0,C 180,E1 -15217.616,E2 -15217.616} C_VEL
LIN {X 0,Y 318.529,Z 758.193,A -85,B 0,C 180,E1 -15219.847,E2 -15219.847} C_VEL
LIN {X 0,Y 319.087,Z 751.058,A -85,B 0,C 180,E1 -15221.757,E2 -15221.757} C_VEL
LIN {X 0,Y 319.886,Z 742.16,A -85,B 0,C 180,E1 -15223.662,E2 -15223.662} C_VEL
LIN {X 0,Y 320.65,Z 734.995,A -85,B 0,C 180,E1 -15224.925,E2 -15224.925} C_VEL
LIN {X 0,Y 321.722,Z 724.23,A -85,B 0,C 180,E1 -15226.499,E2 -15226.499} C_VEL
LIN {X 0,Y 322.921,Z 712.011,A -85,B 0,C 180,E1 -15227.904,E2 -15227.904} C_VEL
LIN {X 0,Y 323.249,Z 707.138,A -85,B 0,C 180,E1 -15228.377,E2 -15228.377} C_VEL
LIN {X 0,Y 322.905,Z 694.754,A -85,B 0,C 180,E1 -15229.418,E2 -15229.418} C_VEL
LIN {X 0,Y 322.046,Z 680.367,A -85,B 0,C 180,E1 -15230.332,E2 -15230.332} C_VEL
LIN {X 0,Y 319.726,Z 656.29,A -85,B 0,C 180,E1 -15231.436,E2 -15231.436} C_VEL
LIN {X 0,Y 319.244,Z 648.879,A -85,B 0,C 180,E1 -15232.123,E2 -15232.123} C_VEL
LIN {X 0,Y 320.155,Z 635.803,A -85,B 0,C 180,E1 -15236.746,E2 -15236.746} C_VEL
LIN {X 0,Y 321.084,Z 626.105,A -85,B 0,C 180,E1 -15240.228,E2 -15240.228} C_VEL
LIN {X 0,Y 322.264,Z 615.671,A -85,B 0,C 180,E1 -15244.033,E2 -15244.033} C_VEL
LIN {X 0,Y 323.369,Z 606.357,A -85,B 0,C 180,E1 -15247.485,E2 -15247.485} C_VEL
LIN {X 0,Y 322.962,Z 602.189,A -85,B 0,C 180,E1 -15249.13,E2 -15249.13} C_VEL
LIN {X 0,Y 321.116,Z 592.455,A -85,B 0,C 180,E1 -15253.201,E2 -15253.201} C_VEL
LIN {X 0,Y 319.558,Z 584.682,A -85,B 0,C 180,E1 -15256.703,E2 -15256.703} C_VEL
LIN {X 0,Y 319.553,Z 584.683,A -85,B 0,C 180,E1 -15260.371,E2 -15260.371} C_VEL
LIN {X 0,Y 319.565,Z 584.678,A -85,B 0,C 180,E1 -15263.573,E2 -15263.573} C_VEL
LIN {X 0,Y 319.583,Z 584.677,A -85,B 0,C 180,E1 -15266.686,E2 -15266.686} C_VEL
LIN {X 0,Y 319.597,Z 584.672,A -85,B 0,C 180,E1 -15269.617,E2 -15269.617} C_VEL
LIN {X 0,Y 319.612,Z 584.674,A -85,B 0,C 180,E1 -15272.498,E2 -15272.498} C_VEL
LIN {X 0,Y 319.61,Z 584.67,A -85,B 0,C 180,E1 -15275.304,E2 -15275.304} C_VEL
LIN {X 0,Y 319.602,Z 584.674,A -85,B 0,C 180,E1 -15278.048,E2 -15278.048} C_VEL
LIN {X 0,Y 319.694,Z 584.661,A -85,B 0,C 180,E1 -15280.962,E2 -15280.962} C_VEL
LIN {X 0,Y 319.736,Z 584.655,A -85,B 0,C 180,E1 -15285.276,E2 -15285.276} C_VEL
LIN {X 0,Y 319.763,Z 584.653,A -85,B 0,C 180,E1 -15289.873,E2 -15289.873} C_VEL
LIN {X 0,Y 319.939,Z 584.634,A -85,B 0,C 180,E1 -15292.426,E2 -15292.426} C_VEL
LIN {X 0,Y 319.75,Z 584.653,A -85,B 0,C 180,E1 -15294.956,E2 -15294.956} C_VEL
LIN {X 0,Y 319.993,Z 584.622,A -85,B 0,C 180,E1 -15297.482,E2 -15297.482} C_VEL
LIN {X 0,Y 320.155,Z 584.604,A -85,B 0,C 180,E1 -15300,E2 -15300} C_VEL
LIN {X 0,Y 319.993,Z 584.625,A -85,B 0,C 180,E1 -15302.517,E2 -15302.517} C_VEL
LIN {X 0,Y 319.935,Z 584.629,A -85,B 0,C 180,E1 -15306.651,E2 -15306.651} C_VEL
LIN {X 0,Y 319.762,Z 584.654,A -85,B 0,C 180,E1 -15310.127,E2 -15310.127} C_VEL
LIN {X 0,Y 319.735,Z 584.655,A -85,B 0,C 180,E1 -15314.723,E2 -15314.723} C_VEL
LIN {X 0,Y 319.693,Z 584.66,A -85,B 0,C 180,E1 -15319.037,E2 -15319.037} C_VEL
LIN {X 0,Y 319.573,Z 584.674,A -85,B 0,C 180,E1 -15323.319,E2 -15323.319} C_VEL
LIN {X 0,Y 319.638,Z 584.667,A -85,B 0,C 180,E1 -15326.087,E2 -15326.087} C_VEL
LIN {X 0,Y 319.592,Z 584.673,A -85,B 0,C 180,E1 -15328.933,E2 -15328.933} C_VEL
LIN {X 0,Y 319.534,Z 584.68,A -85,B 0,C 180,E1 -15331.861,E2 -15331.861} C_VEL
LIN {X 0,Y 319.582,Z 584.673,A -85,B 0,C 180,E1 -15335.542,E2 -15335.542} C_VEL
LIN {X 0,Y 319.559,Z 584.678,A -85,B 0,C 180,E1 -15338.009,E2 -15338.009} C_VEL
LIN {X 0,Y 319.528,Z 584.68,A -85,B 0,C 180,E1 -15341.596,E2 -15341.596} C_VEL
LIN {X 0,Y 319.517,Z 584.683,A -85,B 0,C 180,E1 -15344.737,E2 -15344.737} C_VEL
LIN {X 0,Y 319.553,Z 584.681,A -85,B 0,C 180,E1 -15348.397,E2 -15348.397} C_VEL
LIN {X 0,Y 319.579,Z 584.677,A -85,B 0,C 180,E1 -15352.343,E2 -15352.343} C_VEL
LIN {X 0,Y 319.561,Z 584.677,A -85,B 0,C 180,E1 -15355.122,E2 -15355.122} C_VEL
LIN {X 0,Y 319.567,Z 584.676,A -85,B 0,C 180,E1 -15359.058,E2 -15359.058} C_VEL
LIN {X 0,Y 319.606,Z 584.676,A -85,B 0,C 180,E1 -15362.497,E2 -15362.497} C_VEL
LIN {X 0,Y 319.605,Z 584.671,A -85,B 0,C 180,E1 -15365.303,E2 -15365.303} C_VEL
LIN {X 0,Y 319.598,Z 584.672,A -85,B 0,C 180,E1 -15368.047,E2 -15368.047} C_VEL
LIN {X 0,Y 319.689,Z 584.662,A -85,B 0,C 180,E1 -15370.961,E2 -15370.961} C_VEL
LIN {X 0,Y 319.73,Z 584.655,A -85,B 0,C 180,E1 -15375.275,E2 -15375.275} C_VEL
LIN {X 0,Y 319.759,Z 584.652,A -85,B 0,C 180,E1 -15379.872,E2 -15379.872} C_VEL
LIN {X 0,Y 319.959,Z 584.627,A -85,B 0,C 180,E1 -15383.535,E2 -15383.535} C_VEL
LIN {X 0,Y 319.952,Z 584.628,A -85,B 0,C 180,E1 -15383.654,E2 -15383.654} C_VEL
LIN {X 0,Y 323.213,Z 596.16,A -85,B 0,C 180,E1 -15384.696,E2 -15384.696} C_VEL
LIN {X 0,Y 326.232,Z 606.902,A -85,B 0,C 180,E1 -15385.884,E2 -15385.884} C_VEL
LIN {X 0,Y 325.393,Z 617.321,A -85,B 0,C 180,E1 -15387.059,E2 -15387.059} C_VEL
LIN {X 0,Y 324.5,Z 627.205,A -85,B 0,C 180,E1 -15388.448,E2 -15388.448} C_VEL
LIN {X 0,Y 323.484,Z 636.199,A -85,B 0,C 180,E1 -15389.999,E2 -15389.999} C_VEL
LIN {X 0,Y 322.491,Z 644.966,A -85,B 0,C 180,E1 -15391.872,E2 -15391.872} C_VEL
LIN {X 0,Y 321.713,Z 652.005,A -85,B 0,C 180,E1 -15393.756,E2 -15393.756} C_VEL
LIN {X 0,Y 321.016,Z 657.644,A -85,B 0,C 180,E1 -15395.653,E2 -15395.653} C_VEL
LIN {X 0,Y 320.489,Z 662.096,A -85,B 0,C 180,E1 -15397.559,E2 -15397.559} C_VEL
LIN {X 0,Y 320.166,Z 664.679,A -85,B 0,C 180,E1 -15398.963,E2 -15398.963} C_VEL
LIN {X 0,Y 320.015,Z 666.401,A -85,B 0,C 180,E1 -15400.118,E2 -15400.118} C_VEL
LIN {X 0,Y 319.908,Z 667.885,A -85,B 0,C 180,E1 -15401.402,E2 -15401.402} C_VEL
LIN {X 0,Y 319.89,Z 669.619,A -85,B 0,C 180,E1 -15403.984,E2 -15403.984} C_VEL
LIN {X 0,Y 319.995,Z 669.899,A -85,B 0,C 180,E1 -15405.28,E2 -15405.28} C_VEL
LIN {X 0,Y 320.161,Z 669.733,A -85,B 0,C 180,E1 -15406.58,E2 -15406.58} C_VEL
LIN {X 0,Y 320.399,Z 669.17,A -85,B 0,C 180,E1 -15407.883,E2 -15407.883} C_VEL
LIN {X 0,Y 320.876,Z 667.747,A -85,B 0,C 180,E1 -15409.644,E2 -15409.644} C_VEL
LIN {X 0,Y 321.697,Z 664.901,A -85,B 0,C 180,E1 -15411.8,E2 -15411.8} C_VEL
LIN {X 0,Y 322.628,Z 661.093,A -85,B 0,C 180,E1 -15413.808,E2 -15413.808} C_VEL
LIN {X 0,Y 323.744,Z 656.257,A -85,B 0,C 180,E1 -15415.731,E2 -15415.731} C_VEL
LIN {X 0,Y 325.172,Z 649.606,A -85,B 0,C 180,E1 -15417.784,E2 -15417.784} C_VEL
LIN {X 0,Y 326.697,Z 641.86,A -85,B 0,C 180,E1 -15419.654,E2 -15419.654} C_VEL
LIN {X 0,Y 328.383,Z 632.674,A -85,B 0,C 180,E1 -15421.424,E2 -15421.424} C_VEL
LIN {X 0,Y 329.776,Z 623.062,A -85,B 0,C 180,E1 -15422.917,E2 -15422.917} C_VEL
LIN {X 0,Y 330.725,Z 616.032,A -85,B 0,C 180,E1 -15423.818,E2 -15423.818} C_VEL
LIN {X 0,Y 328.373,Z 607.233,A -85,B 0,C 180,E1 -15425.105,E2 -15425.105} C_VEL
LIN {X 0,Y 325.015,Z 597.699,A -85,B 0,C 180,E1 -15426.381,E2 -15426.381} C_VEL
LIN {X 0,Y 322.649,Z 593.733,A -85,B 0,C 180,E1 -15426.955,E2 -15426.955} C_VEL
LIN {X 0,Y 321.199,Z 591.793,A -85,B 0,C 180,E1 -15427.261,E2 -15427.261} C_VEL
LIN {X 0,Y 320.671,Z 590.4,A -85,B 0,C 180,E1 -15427.454,E2 -15427.454} C_VEL
LIN {X 0,Y 321.504,Z 595.899,A -85,B 0,C 180,E1 -15430.086,E2 -15430.086} C_VEL
LIN {X 0,Y 321.588,Z 600.036,A -85,B 0,C 180,E1 -15432.01,E2 -15432.01} C_VEL
LIN {X 0,Y 321.227,Z 607.868,A -85,B 0,C 180,E1 -15435.564,E2 -15435.564} C_VEL
LIN {X 0,Y 320.729,Z 616.711,A -85,B 0,C 180,E1 -15439.559,E2 -15439.559} C_VEL
LIN {X 0,Y 320.367,Z 624.144,A -85,B 0,C 180,E1 -15442.903,E2 -15442.903} C_VEL
LIN {X 0,Y 320.083,Z 630.821,A -85,B 0,C 180,E1 -15445.889,E2 -15445.889} C_VEL
LIN {X 0,Y 323.121,Z 647.089,A -85,B 0,C 180,E1 -15446.824,E2 -15446.824} C_VEL
LIN {X 0,Y 325.119,Z 658.567,A -85,B 0,C 180,E1 -15447.683,E2 -15447.683} C_VEL
LIN {X 0,Y 324.377,Z 670.281,A -85,B 0,C 180,E1 -15448.669,E2 -15448.669} C_VEL
LIN {X 0,Y 323.195,Z 682.732,A -85,B 0,C 180,E1 -15449.991,E2 -15449.991} C_VEL
LIN {X 0,Y 323.067,Z 684.138,A -85,B 0,C 180,E1 -15450.166,E2 -15450.166} C_VEL
LIN {X 0,Y 321.963,Z 688.916,A -85,B 0,C 180,E1 -15450.76,E2 -15450.76} C_VEL
LIN {X 0,Y 318.357,Z 696.349,A -85,B 0,C 180,E1 -15451.749,E2 -15451.749} C_VEL
LIN {X 0,Y 314.751,Z 703.323,A -85,B 0,C 180,E1 -15452.849,E2 -15452.849} C_VEL
LIN {X 0,Y 313.662,Z 707.335,A -85,B 0,C 180,E1 -15453.607,E2 -15453.607} C_VEL
LIN {X 0,Y 312.723,Z 715.483,A -85,B 0,C 180,E1 -15455.433,E2 -15455.433} C_VEL
LIN {X 0,Y 312.045,Z 722.789,A -85,B 0,C 180,E1 -15457.488,E2 -15457.488} C_VEL
LIN {X 0,Y 311.45,Z 728.551,A -85,B 0,C 180,E1 -15459.528,E2 -15459.528} C_VEL
LIN {X 0,Y 311.133,Z 733.001,A -85,B 0,C 180,E1 -15461.565,E2 -15461.565} C_VEL
LIN {X 0,Y 310.934,Z 735.267,A -85,B 0,C 180,E1 -15462.913,E2 -15462.913} C_VEL
LIN {X 0,Y 310.802,Z 737.064,A -85,B 0,C 180,E1 -15464.256,E2 -15464.256} C_VEL
LIN {X 0,Y 310.805,Z 739.05,A -85,B 0,C 180,E1 -15466.482,E2 -15466.482} C_VEL
LIN {X 0,Y 310.871,Z 739.728,A -85,B 0,C 180,E1 -15468.261,E2 -15468.261} C_VEL
LIN {X 0,Y 310.98,Z 739.767,A -85,B 0,C 180,E1 -15469.584,E2 -15469.584} C_VEL
LIN {X 0,Y 311.172,Z 739.338,A -85,B 0,C 180,E1 -15470.904,E2 -15470.904} C_VEL
LIN {X 0,Y 311.633,Z 737.939,A -85,B 0,C 180,E1 -15472.87,E2 -15472.87} C_VEL
LIN {X 0,Y 312.432,Z 734.613,A -85,B 0,C 180,E1 -15475.485,E2 -15475.485} C_VEL
LIN {X 0,Y 313.253,Z 730.947,A -85,B 0,C 180,E1 -15477.429,E2 -15477.429} C_VEL
LIN {X 0,Y 314.354,Z 726.166,A -85,B 0,C 180,E1 -15479.36,E2 -15479.36} C_VEL
LIN {X 0,Y 315.731,Z 720.123,A -85,B 0,C 180,E1 -15481.276,E2 -15481.276} C_VEL
LIN {X 0,Y 317.565,Z 712.205,A -85,B 0,C 180,E1 -15483.287,E2 -15483.287} C_VEL
LIN {X 0,Y 319.439,Z 703.572,A -85,B 0,C 180,E1 -15485.049,E2 -15485.049} C_VEL
LIN {X 0,Y 321.501,Z 693.152,A -85,B 0,C 180,E1 -15486.748,E2 -15486.748} C_VEL
LIN {X 0,Y 323.612,Z 681.424,A -85,B 0,C 180,E1 -15488.273,E2 -15488.273} C_VEL
LIN {X 0,Y 325.421,Z 669.829,A -85,B 0,C 180,E1 -15489.472,E2 -15489.472} C_VEL
LIN {X 0,Y 325.483,Z 667.344,A -85,B 0,C 180,E1 -15489.729,E2 -15489.729} C_VEL
LIN {X 0,Y 323.895,Z 658.17,A -85,B 0,C 180,E1 -15490.807,E2 -15490.807} C_VEL
LIN {X 0,Y 320.484,Z 646.033,A -85,B 0,C 180,E1 -15492.218,E2 -15492.218} C_VEL
LIN {X 0,Y 316.726,Z 636.147,A -85,B 0,C 180,E1 -15493.401,E2 -15493.401} C_VEL
LIN {X 0,Y 317.729,Z 627.987,A -85,B 0,C 180,E1 -15497.577,E2 -15497.577} C_VEL
LIN {X 0,Y 318.831,Z 620.829,A -85,B 0,C 180,E1 -15501.329,E2 -15501.329} C_VEL
LIN {X 0,Y 319.629,Z 615.975,A -85,B 0,C 180,E1 -15504.003,E2 -15504.003} C_VEL
LIN {X 0,Y 319.669,Z 612.519,A -85,B 0,C 180,E1 -15506.086,E2 -15506.086} C_VEL
LIN {X 0,Y 319.275,Z 608.508,A -85,B 0,C 180,E1 -15508.965,E2 -15508.965} C_VEL
LIN {X 0,Y 318.744,Z 605.15,A -85,B 0,C 180,E1 -15511.95,E2 -15511.95} C_VEL
LIN {X 0,Y 318.187,Z 602.082,A -85,B 0,C 180,E1 -15515.193,E2 -15515.193} C_VEL
LIN {X 0,Y 317.772,Z 600.065,A -85,B 0,C 180,E1 -15518.263,E2 -15518.263} C_VEL
LIN {X 0,Y 317.623,Z 599.429,A -85,B 0,C 180,E1 -15519.918,E2 -15519.918} C_VEL
LIN {X 0,Y 317.268,Z 599.33,A -85,B 0,C 180,E1 -15521.648,E2 -15521.648} C_VEL
LIN {X 0,Y 316.388,Z 600.368,A -85,B 0,C 180,E1 -15524.7,E2 -15524.7} C_VEL
LIN {X 0,Y 316.058,Z 602.072,A -85,B 0,C 180,E1 -15526.816,E2 -15526.816} C_VEL
LIN {X 0,Y 317.588,Z 610.457,A -85,B 0,C 180,E1 -15530.763,E2 -15530.763} C_VEL
LIN {X 0,Y 317.619,Z 614.224,A -85,B 0,C 180,E1 -15532.377,E2 -15532.377} C_VEL
LIN {X 0,Y 315.939,Z 623.789,A -85,B 0,C 180,E1 -15536.214,E2 -15536.214} C_VEL
LIN {X 0,Y 315.116,Z 629.761,A -85,B 0,C 180,E1 -15538.505,E2 -15538.505} C_VEL
LIN {X 0,Y 315.453,Z 639.138,A -85,B 0,C 180,E1 -15540.652,E2 -15540.652} C_VEL
LIN {X 0,Y 316.209,Z 649.809,A -85,B 0,C 180,E1 -15542.753,E2 -15542.753} C_VEL
LIN {X 0,Y 316.645,Z 654.777,A -85,B 0,C 180,E1 -15543.58,E2 -15543.58} C_VEL
LIN {X 0,Y 320.305,Z 669.651,A -85,B 0,C 180,E1 -15544.87,E2 -15544.87} C_VEL
LIN {X 0,Y 321.986,Z 682.113,A -85,B 0,C 180,E1 -15545.907,E2 -15545.907} C_VEL
LIN {X 0,Y 322.061,Z 694.709,A -85,B 0,C 180,E1 -15546.996,E2 -15546.996} C_VEL
LIN {X 0,Y 321.311,Z 706.509,A -85,B 0,C 180,E1 -15548.172,E2 -15548.172} C_VEL
LIN {X 0,Y 320.429,Z 716.033,A -85,B 0,C 180,E1 -15549.289,E2 -15549.289} C_VEL
LIN {X 0,Y 318.347,Z 727.417,A -85,B 0,C 180,E1 -15550.83,E2 -15550.83} C_VEL
LIN {X 0,Y 316.62,Z 735.946,A -85,B 0,C 180,E1 -15552.231,E2 -15552.231} C_VEL
LIN {X 0,Y 314.779,Z 745.209,A -85,B 0,C 180,E1 -15554.078,E2 -15554.078} C_VEL
LIN {X 0,Y 313.464,Z 753.154,A -85,B 0,C 180,E1 -15556.055,E2 -15556.055} C_VEL
LIN {X 0,Y 312.106,Z 760.413,A -85,B 0,C 180,E1 -15558.309,E2 -15558.309} C_VEL
LIN {X 0,Y 311.488,Z 765.297,A -85,B 0,C 180,E1 -15560.259,E2 -15560.259} C_VEL
LIN {X 0,Y 311.089,Z 769.097,A -85,B 0,C 180,E1 -15562.211,E2 -15562.211} C_VEL
LIN {X 0,Y 310.932,Z 771.687,A -85,B 0,C 180,E1 -15564.01,E2 -15564.01} C_VEL
LIN {X 0,Y 310.924,Z 773.69,A -85,B 0,C 180,E1 -15566.113,E2 -15566.113} C_VEL
LIN {X 0,Y 310.919,Z 774.387,A -85,B 0,C 180,E1 -15567.41,E2 -15567.41} C_VEL
LIN {X 0,Y 311.078,Z 774.629,A -85,B 0,C 180,E1 -15568.707,E2 -15568.707} C_VEL
LIN {X 0,Y 311.184,Z 774.451,A -85,B 0,C 180,E1 -15570.001,E2 -15570.001} C_VEL
LIN {X 0,Y 311.163,Z 773.854,A -85,B 0,C 180,E1 -15571.295,E2 -15571.295} C_VEL
LIN {X 0,Y 311.009,Z 772.795,A -85,B 0,C 180,E1 -15572.592,E2 -15572.592} C_VEL
LIN {X 0,Y 310.969,Z 771.269,A -85,B 0,C 180,E1 -15573.889,E2 -15573.889} C_VEL
LIN {X 0,Y 311.043,Z 767.473,A -85,B 0,C 180,E1 -15576.181,E2 -15576.181} C_VEL
LIN {X 0,Y 311.202,Z 762.144,A -85,B 0,C 180,E1 -15578.442,E2 -15578.442} C_VEL
LIN {X 0,Y 311.645,Z 755.016,A -85,B 0,C 180,E1 -15580.723,E2 -15580.723} C_VEL
LIN {X 0,Y 312.384,Z 747.204,A -85,B 0,C 180,E1 -15582.672,E2 -15582.672} C_VEL
LIN {X 0,Y 313.191,Z 739.218,A -85,B 0,C 180,E1 -15584.292,E2 -15584.292} C_VEL
LIN {X 0,Y 314.101,Z 729.735,A -85,B 0,C 180,E1 -15585.875,E2 -15585.875} C_VEL
LIN {X 0,Y 315.242,Z 718.785,A -85,B 0,C 180,E1 -15587.35,E2 -15587.35} C_VEL
LIN {X 0,Y 316.258,Z 708.479,A -85,B 0,C 180,E1 -15588.463,E2 -15588.463} C_VEL
LIN {X 0,Y 315.949,Z 695.779,A -85,B 0,C 180,E1 -15589.596,E2 -15589.596} C_VEL
LIN {X 0,Y 315.24,Z 682.393,A -85,B 0,C 180,E1 -15590.5,E2 -15590.5} C_VEL
LIN {X 0,Y 314.067,Z 668.706,A -85,B 0,C 180,E1 -15591.174,E2 -15591.174} C_VEL
LIN {X 0,Y 312.7,Z 655.393,A -85,B 0,C 180,E1 -15591.855,E2 -15591.855} C_VEL
LIN {X 0,Y 312.201,Z 647.741,A -85,B 0,C 180,E1 -15592.59,E2 -15592.59} C_VEL
LIN {X 0,Y 313.037,Z 636.468,A -85,B 0,C 180,E1 -15596.682,E2 -15596.682} C_VEL
LIN {X 0,Y 314.001,Z 626.822,A -85,B 0,C 180,E1 -15600.239,E2 -15600.239} C_VEL
LIN {X 0,Y 315.338,Z 615.566,A -85,B 0,C 180,E1 -15604.449,E2 -15604.449} C_VEL
LIN {X 0,Y 316.376,Z 607.126,A -85,B 0,C 180,E1 -15607.655,E2 -15607.655} C_VEL
LIN {X 0,Y 315.801,Z 602.606,A -85,B 0,C 180,E1 -15609.501,E2 -15609.501} C_VEL
LIN {X 0,Y 314.128,Z 593.691,A -85,B 0,C 180,E1 -15613.315,E2 -15613.315} C_VEL
LIN {X 0,Y 312.53,Z 585.557,A -85,B 0,C 180,E1 -15617.045,E2 -15617.045} C_VEL
LIN {X 0,Y 312.514,Z 585.557,A -85,B 0,C 180,E1 -15620.973,E2 -15620.973} C_VEL
LIN {X 0,Y 312.538,Z 585.558,A -85,B 0,C 180,E1 -15624.221,E2 -15624.221} C_VEL
LIN {X 0,Y 312.51,Z 585.556,A -85,B 0,C 180,E1 -15627.334,E2 -15627.334} C_VEL
LIN {X 0,Y 312.556,Z 585.549,A -85,B 0,C 180,E1 -15631.277,E2 -15631.277} C_VEL
LIN {X 0,Y 312.591,Z 585.547,A -85,B 0,C 180,E1 -15634.711,E2 -15634.711} C_VEL
LIN {X 0,Y 312.593,Z 585.544,A -85,B 0,C 180,E1 -15637.529,E2 -15637.529} C_VEL
LIN {X 0,Y 312.643,Z 585.539,A -85,B 0,C 180,E1 -15641.656,E2 -15641.656} C_VEL
LIN {X 0,Y 312.699,Z 585.532,A -85,B 0,C 180,E1 -15645.686,E2 -15645.686} C_VEL
LIN {X 0,Y 312.707,Z 585.531,A -85,B 0,C 180,E1 -15649.642,E2 -15649.642} C_VEL
LIN {X 0,Y 312.879,Z 585.513,A -85,B 0,C 180,E1 -15652.254,E2 -15652.254} C_VEL
LIN {X 0,Y 312.721,Z 585.53,A -85,B 0,C 180,E1 -15654.842,E2 -15654.842} C_VEL
LIN {X 0,Y 312.995,Z 585.497,A -85,B 0,C 180,E1 -15658.713,E2 -15658.713} C_VEL
LIN {X 0,Y 312.995,Z 585.493,A -85,B 0,C 180,E1 -15661.286,E2 -15661.286} C_VEL
LIN {X 0,Y 312.72,Z 585.525,A -85,B 0,C 180,E1 -15665.157,E2 -15665.157} C_VEL
LIN {X 0,Y 312.876,Z 585.508,A -85,B 0,C 180,E1 -15667.745,E2 -15667.745} C_VEL
LIN {X 0,Y 312.673,Z 585.534,A -85,B 0,C 180,E1 -15671.671,E2 -15671.671} C_VEL
LIN {X 0,Y 312.704,Z 585.529,A -85,B 0,C 180,E1 -15674.887,E2 -15674.887} C_VEL
LIN {X 0,Y 312.634,Z 585.538,A -85,B 0,C 180,E1 -15679.236,E2 -15679.236} C_VEL
LIN {X 0,Y 312.549,Z 585.551,A -85,B 0,C 180,E1 -15682.788,E2 -15682.788} C_VEL
LIN {X 0,Y 312.606,Z 585.542,A -85,B 0,C 180,E1 -15685.935,E2 -15685.935} C_VEL
LIN {X 0,Y 312.548,Z 585.549,A -85,B 0,C 180,E1 -15689.649,E2 -15689.649} C_VEL
LIN {X 0,Y 312.522,Z 585.553,A -85,B 0,C 180,E1 -15693.688,E2 -15693.688} C_VEL
LIN {X 0,Y 312.528,Z 585.552,A -85,B 0,C 180,E1 -15697.384,E2 -15697.384} C_VEL
LIN {X 0,Y 312.492,Z 585.56,A -85,B 0,C 180,E1 -15700.708,E2 -15700.708} C_VEL
LIN {X 0,Y 312.475,Z 585.56,A -85,B 0,C 180,E1 -15704.205,E2 -15704.205} C_VEL
LIN {X 0,Y 312.516,Z 585.554,A -85,B 0,C 180,E1 -15707.911,E2 -15707.911} C_VEL
LIN {X 0,Y 312.536,Z 585.55,A -85,B 0,C 180,E1 -15711.909,E2 -15711.909} C_VEL
LIN {X 0,Y 312.507,Z 585.555,A -85,B 0,C 180,E1 -15715.789,E2 -15715.789} C_VEL
LIN {X 0,Y 312.521,Z 585.555,A -85,B 0,C 180,E1 -15718.853,E2 -15718.853} C_VEL
LIN {X 0,Y 312.57,Z 585.547,A -85,B 0,C 180,E1 -15721.823,E2 -15721.823} C_VEL
LIN {X 0,Y 312.585,Z 585.549,A -85,B 0,C 180,E1 -15724.71,E2 -15724.71} C_VEL
LIN {X 0,Y 312.588,Z 585.544,A -85,B 0,C 180,E1 -15727.528,E2 -15727.528} C_VEL
LIN {X 0,Y 312.638,Z 585.539,A -85,B 0,C 180,E1 -15731.655,E2 -15731.655} C_VEL
LIN {X 0,Y 312.694,Z 585.531,A -85,B 0,C 180,E1 -15735.685,E2 -15735.685} C_VEL
LIN {X 0,Y 312.703,Z 585.531,A -85,B 0,C 180,E1 -15739.641,E2 -15739.641} C_VEL
LIN {X 0,Y 312.915,Z 585.505,A -85,B 0,C 180,E1 -15743.268,E2 -15743.268} C_VEL
LIN {X 0,Y 316.603,Z 598.388,A -85,B 0,C 180,E1 -15744.474,E2 -15744.474} C_VEL
LIN {X 0,Y 319.139,Z 607.374,A -85,B 0,C 180,E1 -15745.502,E2 -15745.502} C_VEL
LIN {X 0,Y 319.234,Z 610.294,A -85,B 0,C 180,E1 -15745.827,E2 -15745.827} C_VEL
LIN {X 0,Y 318.271,Z 621.134,A -85,B 0,C 180,E1 -15747.151,E2 -15747.151} C_VEL
LIN {X 0,Y 317.262,Z 631.48,A -85,B 0,C 180,E1 -15748.73,E2 -15748.73} C_VEL
LIN {X 0,Y 316.261,Z 639.759,A -85,B 0,C 180,E1 -15750.285,E2 -15750.285} C_VEL
LIN {X 0,Y 315.301,Z 648.098,A -85,B 0,C 180,E1 -15752.234,E2 -15752.234} C_VEL
LIN {X 0,Y 314.543,Z 654.711,A -85,B 0,C 180,E1 -15754.163,E2 -15754.163} C_VEL
LIN {X 0,Y 313.752,Z 660.8,A -85,B 0,C 180,E1 -15756.429,E2 -15756.429} C_VEL
LIN {X 0,Y 313.272,Z 664.766,A -85,B 0,C 180,E1 -15758.384,E2 -15758.384} C_VEL
LIN {X 0,Y 312.953,Z 667.707,A -85,B 0,C 180,E1 -15760.348,E2 -15760.348} C_VEL
LIN {X 0,Y 312.853,Z 669.105,A -85,B 0,C 180,E1 -15761.663,E2 -15761.663} C_VEL
LIN {X 0,Y 312.882,Z 670.73,A -85,B 0,C 180,E1 -15764.304,E2 -15764.304} C_VEL
LIN {X 0,Y 313.019,Z 670.903,A -85,B 0,C 180,E1 -15765.629,E2 -15765.629} C_VEL
LIN {X 0,Y 313.48,Z 670.062,A -85,B 0,C 180,E1 -15768.291,E2 -15768.291} C_VEL
LIN {X 0,Y 313.947,Z 668.71,A -85,B 0,C 180,E1 -15769.915,E2 -15769.915} C_VEL
LIN {X 0,Y 314.924,Z 665.559,A -85,B 0,C 180,E1 -15772.294,E2 -15772.294} C_VEL
LIN {X 0,Y 315.853,Z 661.974,A -85,B 0,C 180,E1 -15774.178,E2 -15774.178} C_VEL
LIN {X 0,Y 317.147,Z 656.642,A -85,B 0,C 180,E1 -15776.307,E2 -15776.307} C_VEL
LIN {X 0,Y 318.565,Z 650.121,A -85,B 0,C 180,E1 -15778.308,E2 -15778.308} C_VEL
LIN {X 0,Y 320.31,Z 641.832,A -85,B 0,C 180,E1 -15780.306,E2 -15780.306} C_VEL
LIN {X 0,Y 321.906,Z 633.244,A -85,B 0,C 180,E1 -15781.966,E2 -15781.966} C_VEL
LIN {X 0,Y 323.396,Z 623.737,A -85,B 0,C 180,E1 -15783.449,E2 -15783.449} C_VEL
LIN {X 0,Y 324.124,Z 617.254,A -85,B 0,C 180,E1 -15784.314,E2 -15784.314} C_VEL
LIN {X 0,Y 321.56,Z 608.289,A -85,B 0,C 180,E1 -15785.686,E2 -15785.686} C_VEL
LIN {X 0,Y 318.735,Z 600.535,A -85,B 0,C 180,E1 -15786.78,E2 -15786.78} C_VEL
LIN {X 0,Y 314,Z 593.326,A -85,B 0,C 180,E1 -15787.92,E2 -15787.92} C_VEL
LIN {X 0,Y 313.927,Z 592.988,A -85,B 0,C 180,E1 -15787.992,E2 -15787.992} C_VEL
LIN {X 0,Y 314.622,Z 598.396,A -85,B 0,C 180,E1 -15790.582,E2 -15790.582} C_VEL
LIN {X 0,Y 314.514,Z 603.826,A -85,B 0,C 180,E1 -15793.109,E2 -15793.109} C_VEL
LIN {X 0,Y 314.053,Z 612.133,A -85,B 0,C 180,E1 -15796.926,E2 -15796.926} C_VEL
LIN {X 0,Y 313.572,Z 621.377,A -85,B 0,C 180,E1 -15801.131,E2 -15801.131} C_VEL
LIN {X 0,Y 313.168,Z 630.131,A -85,B 0,C 180,E1 -15805.093,E2 -15805.093} C_VEL
LIN {X 0,Y 313.093,Z 631.179,A -85,B 0,C 180,E1 -15805.569,E2 -15805.569} C_VEL
LIN {X 0,Y 315.913,Z 646.35,A -85,B 0,C 180,E1 -15806.443,E2 -15806.443} C_VEL
LIN {X 0,Y 318.073,Z 658.832,A -85,B 0,C 180,E1 -15807.39,E2 -15807.39} C_VEL
LIN {X 0,Y 317.721,Z 667.516,A -85,B 0,C 180,E1 -15808.122,E2 -15808.122} C_VEL
LIN {X 0,Y 316.62,Z 679.196,A -85,B 0,C 180,E1 -15809.302,E2 -15809.302} C_VEL
LIN {X 0,Y 315.414,Z 691.09,A -85,B 0,C 180,E1 -15810.83,E2 -15810.83} C_VEL
LIN {X 0,Y 314.387,Z 700.771,A -85,B 0,C 180,E1 -15812.364,E2 -15812.364} C_VEL
LIN {X 0,Y 313.662,Z 707.335,A -85,B 0,C 180,E1 -15813.607,E2 -15813.607} C_VEL
LIN {X 0,Y 312.608,Z 711.209,A -85,B 0,C 180,E1 -15814.4,E2 -15814.4} C_VEL
LIN {X 0,Y 309.155,Z 717.054,A -85,B 0,C 180,E1 -15815.732,E2 -15815.732} C_VEL
LIN {X 0,Y 305.736,Z 722.287,A -85,B 0,C 180,E1 -15817.174,E2 -15817.174} C_VEL
LIN {X 0,Y 304.757,Z 725.204,A -85,B 0,C 180,E1 -15818.125,E2 -15818.125} C_VEL
LIN {X 0,Y 304.227,Z 731.022,A -85,B 0,C 180,E1 -15820.43,E2 -15820.43} C_VEL
LIN {X 0,Y 303.897,Z 734.946,A -85,B 0,C 180,E1 -15822.504,E2 -15822.504} C_VEL
LIN {X 0,Y 303.729,Z 736.917,A -85,B 0,C 180,E1 -15823.879,E2 -15823.879} C_VEL
LIN {X 0,Y 303.718,Z 739.301,A -85,B 0,C 180,E1 -15826.372,E2 -15826.372} C_VEL
LIN {X 0,Y 303.781,Z 740.072,A -85,B 0,C 180,E1 -15827.983,E2 -15827.983} C_VEL
LIN {X 0,Y 303.863,Z 740.238,A -85,B 0,C 180,E1 -15829.338,E2 -15829.338} C_VEL
LIN {X 0,Y 304.058,Z 740.002,A -85,B 0,C 180,E1 -15830.689,E2 -15830.689} C_VEL
LIN {X 0,Y 304.573,Z 738.743,A -85,B 0,C 180,E1 -15832.835,E2 -15832.835} C_VEL
LIN {X 0,Y 305.072,Z 736.743,A -85,B 0,C 180,E1 -15834.713,E2 -15834.713} C_VEL
LIN {X 0,Y 305.843,Z 733.671,A -85,B 0,C 180,E1 -15836.707,E2 -15836.707} C_VEL
LIN {X 0,Y 306.934,Z 729.546,A -85,B 0,C 180,E1 -15838.688,E2 -15838.688} C_VEL
LIN {X 0,Y 308.46,Z 723.321,A -85,B 0,C 180,E1 -15840.98,E2 -15840.98} C_VEL
LIN {X 0,Y 310.18,Z 716.397,A -85,B 0,C 180,E1 -15842.959,E2 -15842.959} C_VEL
LIN {X 0,Y 312.166,Z 708.182,A -85,B 0,C 180,E1 -15844.844,E2 -15844.844} C_VEL
LIN {X 0,Y 314.452,Z 697.835,A -85,B 0,C 180,E1 -15846.739,E2 -15846.739} C_VEL
LIN {X 0,Y 316.641,Z 687.198,A -85,B 0,C 180,E1 -15848.296,E2 -15848.296} C_VEL
LIN {X 0,Y 318.709,Z 675.316,A -85,B 0,C 180,E1 -15849.68,E2 -15849.68} C_VEL
LIN {X 0,Y 319.437,Z 670.657,A -85,B 0,C 180,E1 -15850.138,E2 -15850.138} C_VEL
LIN {X 0,Y 318.304,Z 661.866,A -85,B 0,C 180,E1 -15851.221,E2 -15851.221} C_VEL
LIN {X 0,Y 315.453,Z 650.669,A -85,B 0,C 180,E1 -15852.621,E2 -15852.621} C_VEL
LIN {X 0,Y 311.459,Z 639.944,A -85,B 0,C 180,E1 -15854.01,E2 -15854.01} C_VEL
LIN {X 0,Y 310.25,Z 636.737,A -85,B 0,C 180,E1 -15854.43,E2 -15854.43} C_VEL
LIN {X 0,Y 311.361,Z 628.914,A -85,B 0,C 180,E1 -15858.56,E2 -15858.56} C_VEL
LIN {X 0,Y 312.657,Z 621.792,A -85,B 0,C 180,E1 -15862.466,E2 -15862.466} C_VEL
LIN {X 0,Y 313.228,Z 618.221,A -85,B 0,C 180,E1 -15864.526,E2 -15864.526} C_VEL
LIN {X 0,Y 313.28,Z 614.951,A -85,B 0,C 180,E1 -15866.659,E2 -15866.659} C_VEL
LIN {X 0,Y 312.988,Z 611.296,A -85,B 0,C 180,E1 -15869.604,E2 -15869.604} C_VEL
LIN {X 0,Y 312.473,Z 607.986,A -85,B 0,C 180,E1 -15872.67,E2 -15872.67} C_VEL
LIN {X 0,Y 312.071,Z 605.373,A -85,B 0,C 180,E1 -15875.841,E2 -15875.841} C_VEL
LIN {X 0,Y 311.87,Z 603.734,A -85,B 0,C 180,E1 -15879.123,E2 -15879.123} C_VEL
LIN {X 0,Y 311.694,Z 603.449,A -85,B 0,C 180,E1 -15880.836,E2 -15880.836} C_VEL
LIN {X 0,Y 311.225,Z 603.808,A -85,B 0,C 180,E1 -15882.646,E2 -15882.646} C_VEL
LIN {X 0,Y 310.838,Z 604.654,A -85,B 0,C 180,E1 -15884.5,E2 -15884.5} C_VEL
LIN {X 0,Y 310.31,Z 607.03,A -85,B 0,C 180,E1 -15887.201,E2 -15887.201} C_VEL
LIN {X 0,Y 310.493,Z 610.858,A -85,B 0,C 180,E1 -15890.199,E2 -15890.199} C_VEL
LIN {X 0,Y 310.789,Z 613.826,A -85,B 0,C 180,E1 -15891.549,E2 -15891.549} C_VEL
LIN {X 0,Y 309.894,Z 619.373,A -85,B 0,C 180,E1 -15893.87,E2 -15893.87} C_VEL
LIN {X 0,Y 309.396,Z 623.885,A -85,B 0,C 180,E1 -15895.399,E2 -15895.399} C_VEL
LIN {X 0,Y 309.352,Z 633.744,A -85,B 0,C 180,E1 -15898.208,E2 -15898.208} C_VEL
LIN {X 0,Y 309.659,Z 644.37,A -85,B 0,C 180,E1 -15900.651,E2 -15900.651} C_VEL
LIN {X 0,Y 310.28,Z 653.898,A -85,B 0,C 180,E1 -15902.539,E2 -15902.539} C_VEL
LIN {X 0,Y 314.017,Z 668.841,A -85,B 0,C 180,E1 -15903.948,E2 -15903.948} C_VEL
LIN {X 0,Y 315.841,Z 681.603,A -85,B 0,C 180,E1 -15905.097,E2 -15905.097} C_VEL
LIN {X 0,Y 315.944,Z 694.541,A -85,B 0,C 180,E1 -15906.276,E2 -15906.276} C_VEL
LIN {X 0,Y 315.022,Z 706.96,A -85,B 0,C 180,E1 -15907.556,E2 -15907.556} C_VEL
LIN {X 0,Y 314.143,Z 716.077,A -85,B 0,C 180,E1 -15908.683,E2 -15908.683} C_VEL
LIN {X 0,Y 311.71,Z 728.3,A -85,B 0,C 180,E1 -15910.406,E2 -15910.406} C_VEL
LIN {X 0,Y 309.918,Z 736.624,A -85,B 0,C 180,E1 -15911.833,E2 -15911.833} C_VEL
LIN {X 0,Y 307.923,Z 745.831,A -85,B 0,C 180,E1 -15913.764,E2 -15913.764} C_VEL
LIN {X 0,Y 306.368,Z 754.49,A -85,B 0,C 180,E1 -15916.064,E2 -15916.064} C_VEL
LIN {X 0,Y 305.123,Z 760.476,A -85,B 0,C 180,E1 -15918.037,E2 -15918.037} C_VEL
LIN {X 0,Y 304.446,Z 765.249,A -85,B 0,C 180,E1 -15920.031,E2 -15920.031} C_VEL
LIN {X 0,Y 304.034,Z 768.94,A -85,B 0,C 180,E1 -15922.029,E2 -15922.029} C_VEL
LIN {X 0,Y 303.85,Z 771.641,A -85,B 0,C 180,E1 -15924.038,E2 -15924.038} C_VEL
LIN {X 0,Y 303.827,Z 773.361,A -85,B 0,C 180,E1 -15926.022,E2 -15926.022} C_VEL
LIN {X 0,Y 303.833,Z 773.98,A -85,B 0,C 180,E1 -15927.35,E2 -15927.35} C_VEL
LIN {X 0,Y 303.983,Z 774.173,A -85,B 0,C 180,E1 -15928.676,E2 -15928.676} C_VEL
LIN {X 0,Y 304.124,Z 773.957,A -85,B 0,C 180,E1 -15930.001,E2 -15930.001} C_VEL
LIN {X 0,Y 304.083,Z 773.309,A -85,B 0,C 180,E1 -15931.326,E2 -15931.326} C_VEL
LIN {X 0,Y 303.923,Z 772.169,A -85,B 0,C 180,E1 -15932.652,E2 -15932.652} C_VEL
LIN {X 0,Y 303.918,Z 769.656,A -85,B 0,C 180,E1 -15934.644,E2 -15934.644} C_VEL
LIN {X 0,Y 303.98,Z 766.055,A -85,B 0,C 180,E1 -15936.639,E2 -15936.639} C_VEL
LIN {X 0,Y 304.145,Z 761.265,A -85,B 0,C 180,E1 -15938.64,E2 -15938.64} C_VEL
LIN {X 0,Y 304.547,Z 755.167,A -85,B 0,C 180,E1 -15940.64,E2 -15940.64} C_VEL
LIN {X 0,Y 305.26,Z 747.548,A -85,B 0,C 180,E1 -15942.635,E2 -15942.635} C_VEL
LIN {X 0,Y 306.034,Z 739.704,A -85,B 0,C 180,E1 -15944.294,E2 -15944.294} C_VEL
LIN {X 0,Y 306.992,Z 730.184,A -85,B 0,C 180,E1 -15945.946,E2 -15945.946} C_VEL
LIN {X 0,Y 308.174,Z 719.765,A -85,B 0,C 180,E1 -15947.418,E2 -15947.418} C_VEL
LIN {X 0,Y 309.216,Z 708.111,A -85,B 0,C 180,E1 -15948.727,E2 -15948.727} C_VEL
LIN {X 0,Y 308.961,Z 695.696,A -85,B 0,C 180,E1 -15949.865,E2 -15949.865} C_VEL
LIN {X 0,Y 308.241,Z 682.355,A -85,B 0,C 180,E1 -15950.801,E2 -15950.801} C_VEL
LIN {X 0,Y 307.115,Z 668.63,A -85,B 0,C 180,E1 -15951.501,E2 -15951.501} C_VEL
LIN {X 0,Y 305.646,Z 654.19,A -85,B 0,C 180,E1 -15952.298,E2 -15952.298} C_VEL
LIN {X 0,Y 305.197,Z 646.589,A -85,B 0,C 180,E1 -15953.092,E2 -15953.092} C_VEL
LIN {X 0,Y 306.112,Z 635.255,A -85,B 0,C 180,E1 -15957.335,E2 -15957.335} C_VEL
LIN {X 0,Y 307.115,Z 625.575,A -85,B 0,C 180,E1 -15960.991,E2 -15960.991} C_VEL
LIN {X 0,Y 308.39,Z 615.435,A -85,B 0,C 180,E1 -15964.873,E2 -15964.873} C_VEL
LIN {X 0,Y 309.362,Z 607.868,A -85,B 0,C 180,E1 -15967.835,E2 -15967.835} C_VEL
LIN {X 0,Y 308.473,Z 601.823,A -85,B 0,C 180,E1 -15970.388,E2 -15970.388} C_VEL
LIN {X 0,Y 306.859,Z 593.598,A -85,B 0,C 180,E1 -15974.026,E2 -15974.026} C_VEL
LIN {X 0,Y 305.478,Z 586.434,A -85,B 0,C 180,E1 -15977.411,E2 -15977.411} C_VEL
LIN {X 0,Y 305.501,Z 586.431,A -85,B 0,C 180,E1 -15981.601,E2 -15981.601} C_VEL
LIN {X 0,Y 305.468,Z 586.435,A -85,B 0,C 180,E1 -15984.887,E2 -15984.887} C_VEL
LIN {X 0,Y 305.458,Z 586.439,A -85,B 0,C 180,E1 -15988.355,E2 -15988.355} C_VEL
LIN {X 0,Y 305.525,Z 586.425,A -85,B 0,C 180,E1 -15991.114,E2 -15991.114} C_VEL
LIN {X 0,Y 305.576,Z 586.422,A -85,B 0,C 180,E1 -15994.088,E2 -15994.088} C_VEL
LIN {X 0,Y 305.531,Z 586.429,A -85,B 0,C 180,E1 -15998.405,E2 -15998.405} C_VEL
LIN {X 0,Y 305.595,Z 586.416,A -85,B 0,C 180,E1 -16001.217,E2 -16001.217} C_VEL
LIN {X 0,Y 305.654,Z 586.409,A -85,B 0,C 180,E1 -16005.349,E2 -16005.349} C_VEL
LIN {X 0,Y 305.643,Z 586.41,A -85,B 0,C 180,E1 -16009.399,E2 -16009.399} C_VEL
LIN {X 0,Y 305.82,Z 586.391,A -85,B 0,C 180,E1 -16012.074,E2 -16012.074} C_VEL
LIN {X 0,Y 305.692,Z 586.406,A -85,B 0,C 180,E1 -16014.723,E2 -16014.723} C_VEL
LIN {X 0,Y 305.961,Z 586.373,A -85,B 0,C 180,E1 -16018.683,E2 -16018.683} C_VEL
LIN {X 0,Y 305.961,Z 586.369,A -85,B 0,C 180,E1 -16021.316,E2 -16021.316} C_VEL
LIN {X 0,Y 305.855,Z 586.385,A -85,B 0,C 180,E1 -16026.612,E2 -16026.612} C_VEL
LIN {X 0,Y 305.74,Z 586.398,A -85,B 0,C 180,E1 -16029.259,E2 -16029.259} C_VEL
LIN {X 0,Y 305.592,Z 586.415,A -85,B 0,C 180,E1 -16033.295,E2 -16033.295} C_VEL
LIN {X 0,Y 305.597,Z 586.414,A -85,B 0,C 180,E1 -16036.019,E2 -16036.019} C_VEL
LIN {X 0,Y 305.58,Z 586.417,A -85,B 0,C 180,E1 -16039.444,E2 -16039.444} C_VEL
LIN {X 0,Y 305.493,Z 586.429,A -85,B 0,C 180,E1 -16043.04,E2 -16043.04} C_VEL
LIN {X 0,Y 305.55,Z 586.422,A -85,B 0,C 180,E1 -16046.226,E2 -16046.226} C_VEL
LIN {X 0,Y 305.498,Z 586.428,A -85,B 0,C 180,E1 -16049.049,E2 -16049.049} C_VEL
LIN {X 0,Y 305.467,Z 586.431,A -85,B 0,C 180,E1 -16053.516,E2 -16053.516} C_VEL
LIN {X 0,Y 305.477,Z 586.433,A -85,B 0,C 180,E1 -16056.738,E2 -16056.738} C_VEL
LIN {X 0,Y 305.456,Z 586.437,A -85,B 0,C 180,E1 -16060.599,E2 -16060.599} C_VEL
LIN {X 0,Y 305.421,Z 586.44,A -85,B 0,C 180,E1 -16064.492,E2 -16064.492} C_VEL
LIN {X 0,Y 305.466,Z 586.434,A -85,B 0,C 180,E1 -16068.146,E2 -16068.146} C_VEL
LIN {X 0,Y 305.496,Z 586.426,A -85,B 0,C 180,E1 -16071.599,E2 -16071.599} C_VEL
LIN {X 0,Y 305.464,Z 586.434,A -85,B 0,C 180,E1 -16074.886,E2 -16074.886} C_VEL
LIN {X 0,Y 305.45,Z 586.437,A -85,B 0,C 180,E1 -16078.355,E2 -16078.355} C_VEL
LIN {X 0,Y 305.513,Z 586.427,A -85,B 0,C 180,E1 -16081.112,E2 -16081.112} C_VEL
LIN {X 0,Y 305.565,Z 586.42,A -85,B 0,C 180,E1 -16084.086,E2 -16084.086} C_VEL
LIN {X 0,Y 305.501,Z 586.431,A -85,B 0,C 180,E1 -16088.402,E2 -16088.402} C_VEL
LIN {X 0,Y 305.59,Z 586.418,A -85,B 0,C 180,E1 -16091.217,E2 -16091.217} C_VEL
LIN {X 0,Y 305.649,Z 586.409,A -85,B 0,C 180,E1 -16095.348,E2 -16095.348} C_VEL
LIN {X 0,Y 305.64,Z 586.411,A -85,B 0,C 180,E1 -16099.399,E2 -16099.399} C_VEL
LIN {X 0,Y 305.859,Z 586.387,A -85,B 0,C 180,E1 -16102.863,E2 -16102.863} C_VEL
LIN {X 0,Y 309.231,Z 597.976,A -85,B 0,C 180,E1 -16103.966,E2 -16103.966} C_VEL
LIN {X 0,Y 312.277,Z 608.636,A -85,B 0,C 180,E1 -16105.203,E2 -16105.203} C_VEL
LIN {X 0,Y 312.518,Z 610.37,A -85,B 0,C 180,E1 -16105.407,E2 -16105.407} C_VEL
LIN {X 0,Y 311.491,Z 621.438,A -85,B 0,C 180,E1 -16106.765,E2 -16106.765} C_VEL
LIN {X 0,Y 310.45,Z 631.897,A -85,B 0,C 180,E1 -16108.377,E2 -16108.377} C_VEL
LIN {X 0,Y 309.386,Z 640.451,A -85,B 0,C 180,E1 -16109.999,E2 -16109.999} C_VEL
LIN {X 0,Y 308.407,Z 648.728,A -85,B 0,C 180,E1 -16111.958,E2 -16111.958} C_VEL
LIN {X 0,Y 307.602,Z 655.412,A -85,B 0,C 180,E1 -16113.929,E2 -16113.929} C_VEL
LIN {X 0,Y 306.864,Z 660.789,A -85,B 0,C 180,E1 -16115.914,E2 -16115.914} C_VEL
LIN {X 0,Y 306.333,Z 664.996,A -85,B 0,C 180,E1 -16117.911,E2 -16117.911} C_VEL
LIN {X 0,Y 306.071,Z 667.232,A -85,B 0,C 180,E1 -16119.248,E2 -16119.248} C_VEL
LIN {X 0,Y 305.891,Z 668.983,A -85,B 0,C 180,E1 -16120.59,E2 -16120.59} C_VEL
LIN {X 0,Y 305.819,Z 670.325,A -85,B 0,C 180,E1 -16121.935,E2 -16121.935} C_VEL
LIN {X 0,Y 305.792,Z 671.282,A -85,B 0,C 180,E1 -16123.286,E2 -16123.286} C_VEL
LIN {X 0,Y 305.946,Z 671.899,A -85,B 0,C 180,E1 -16125.25,E2 -16125.25} C_VEL
LIN {X 0,Y 306.27,Z 671.627,A -85,B 0,C 180,E1 -16127.355,E2 -16127.355} C_VEL
LIN {X 0,Y 306.572,Z 670.943,A -85,B 0,C 180,E1 -16128.718,E2 -16128.718} C_VEL
LIN {X 0,Y 307.039,Z 669.666,A -85,B 0,C 180,E1 -16130.205,E2 -16130.205} C_VEL
LIN {X 0,Y 308.142,Z 666.214,A -85,B 0,C 180,E1 -16132.812,E2 -16132.812} C_VEL
LIN {X 0,Y 309.248,Z 662.192,A -85,B 0,C 180,E1 -16134.877,E2 -16134.877} C_VEL
LIN {X 0,Y 310.81,Z 655.964,A -85,B 0,C 180,E1 -16137.249,E2 -16137.249} C_VEL
LIN {X 0,Y 312.397,Z 649.153,A -85,B 0,C 180,E1 -16139.257,E2 -16139.257} C_VEL
LIN {X 0,Y 314.213,Z 640.595,A -85,B 0,C 180,E1 -16141.233,E2 -16141.233} C_VEL
LIN {X 0,Y 315.985,Z 630.912,A -85,B 0,C 180,E1 -16143.017,E2 -16143.017} C_VEL
LIN {X 0,Y 317.634,Z 620.301,A -85,B 0,C 180,E1 -16144.566,E2 -16144.566} C_VEL
LIN {X 0,Y 315.876,Z 612.892,A -85,B 0,C 180,E1 -16145.753,E2 -16145.753} C_VEL
LIN {X 0,Y 313.237,Z 605.005,A -85,B 0,C 180,E1 -16146.937,E2 -16146.937} C_VEL
LIN {X 0,Y 309.081,Z 598.604,A -85,B 0,C 180,E1 -16148.035,E2 -16148.035} C_VEL
LIN {X 0,Y 307.443,Z 596.417,A -85,B 0,C 180,E1 -16148.41,E2 -16148.41} C_VEL
LIN {X 0,Y 307.178,Z 595.575,A -85,B 0,C 180,E1 -16148.529,E2 -16148.529} C_VEL
LIN {X 0,Y 307.716,Z 600.869,A -85,B 0,C 180,E1 -16151.089,E2 -16151.089} C_VEL
LIN {X 0,Y 307.391,Z 607.297,A -85,B 0,C 180,E1 -16154.074,E2 -16154.074} C_VEL
LIN {X 0,Y 306.919,Z 615.179,A -85,B 0,C 180,E1 -16157.736,E2 -16157.736} C_VEL
LIN {X 0,Y 306.471,Z 623.875,A -85,B 0,C 180,E1 -16161.746,E2 -16161.746} C_VEL
LIN {X 0,Y 306.103,Z 631.627,A -85,B 0,C 180,E1 -16165.261,E2 -16165.261} C_VEL
LIN {X 0,Y 308.657,Z 645.62,A -85,B 0,C 180,E1 -16166.055,E2 -16166.055} C_VEL
LIN {X 0,Y 310.987,Z 658.743,A -85,B 0,C 180,E1 -16167.06,E2 -16167.06} C_VEL
LIN {X 0,Y 311.14,Z 663.194,A -85,B 0,C 180,E1 -16167.438,E2 -16167.438} C_VEL
LIN {X 0,Y 310.126,Z 675.282,A -85,B 0,C 180,E1 -16168.586,E2 -16168.586} C_VEL
LIN {X 0,Y 308.891,Z 686.751,A -85,B 0,C 180,E1 -16169.964,E2 -16169.964} C_VEL
LIN {X 0,Y 307.77,Z 697.276,A -85,B 0,C 180,E1 -16171.532,E2 -16171.532} C_VEL
LIN {X 0,Y 306.647,Z 707.522,A -85,B 0,C 180,E1 -16173.435,E2 -16173.435} C_VEL
LIN {X 0,Y 305.732,Z 715.281,A -85,B 0,C 180,E1 -16175.196,E2 -16175.196} C_VEL
LIN {X 0,Y 305.037,Z 722.283,A -85,B 0,C 180,E1 -16177.156,E2 -16177.156} C_VEL
LIN {X 0,Y 304.757,Z 725.204,A -85,B 0,C 180,E1 -16178.125,E2 -16178.125} C_VEL
LIN {X 0,Y 303.814,Z 727.942,A -85,B 0,C 180,E1 -16179.098,E2 -16179.098} C_VEL
LIN {X 0,Y 300.591,Z 731.94,A -85,B 0,C 180,E1 -16180.71,E2 -16180.71} C_VEL
LIN {X 0,Y 297.954,Z 734.598,A -85,B 0,C 180,E1 -16182.058,E2 -16182.058} C_VEL
LIN {X 0,Y 296.784,Z 736.24,A -85,B 0,C 180,E1 -16183.135,E2 -16183.135} C_VEL
LIN {X 0,Y 296.663,Z 736.71,A -85,B 0,C 180,E1 -16183.505,E2 -16183.505} C_VEL
LIN {X 0,Y 296.61,Z 738.375,A -85,B 0,C 180,E1 -16184.893,E2 -16184.893} C_VEL
LIN {X 0,Y 296.624,Z 739.566,A -85,B 0,C 180,E1 -16186.295,E2 -16186.295} C_VEL
LIN {X 0,Y 296.682,Z 740.343,A -85,B 0,C 180,E1 -16187.691,E2 -16187.691} C_VEL
LIN {X 0,Y 296.751,Z 740.704,A -85,B 0,C 180,E1 -16189.079,E2 -16189.079} C_VEL
LIN {X 0,Y 296.945,Z 740.595,A -85,B 0,C 180,E1 -16190.464,E2 -16190.464} C_VEL
LIN {X 0,Y 297.49,Z 739.458,A -85,B 0,C 180,E1 -16192.835,E2 -16192.835} C_VEL
LIN {X 0,Y 297.975,Z 737.824,A -85,B 0,C 180,E1 -16194.587,E2 -16194.587} C_VEL
LIN {X 0,Y 298.778,Z 735.031,A -85,B 0,C 180,E1 -16196.629,E2 -16196.629} C_VEL
LIN {X 0,Y 299.882,Z 731.207,A -85,B 0,C 180,E1 -16198.658,E2 -16198.658} C_VEL
LIN {X 0,Y 301.19,Z 726.279,A -85,B 0,C 180,E1 -16200.669,E2 -16200.669} C_VEL
LIN {X 0,Y 303.219,Z 718.831,A -85,B 0,C 180,E1 -16203.023,E2 -16203.023} C_VEL
LIN {X 0,Y 305.212,Z 711.089,A -85,B 0,C 180,E1 -16204.954,E2 -16204.954} C_VEL
LIN {X 0,Y 307.638,Z 701.375,A -85,B 0,C 180,E1 -16206.889,E2 -16206.889} C_VEL
LIN {X 0,Y 309.84,Z 691.393,A -85,B 0,C 180,E1 -16208.479,E2 -16208.479} C_VEL
LIN {X 0,Y 312.266,Z 679.17,A -85,B 0,C 180,E1 -16210.046,E2 -16210.046} C_VEL
LIN {X 0,Y 313.451,Z 672.196,A -85,B 0,C 180,E1 -16210.78,E2 -16210.78} C_VEL
LIN {X 0,Y 312.4,Z 663.992,A -85,B 0,C 180,E1 -16211.864,E2 -16211.864} C_VEL
LIN {X 0,Y 309.869,Z 653.571,A -85,B 0,C 180,E1 -16213.26,E2 -16213.26} C_VEL
LIN {X 0,Y 306.391,Z 643.791,A -85,B 0,C 180,E1 -16214.615,E2 -16214.615} C_VEL
LIN {X 0,Y 303.893,Z 637.446,A -85,B 0,C 180,E1 -16215.51,E2 -16215.51} C_VEL
LIN {X 0,Y 304.964,Z 630.829,A -85,B 0,C 180,E1 -16219.121,E2 -16219.121} C_VEL
LIN {X 0,Y 306.326,Z 624.059,A -85,B 0,C 180,E1 -16222.957,E2 -16222.957} C_VEL
LIN {X 0,Y 306.918,Z 620.613,A -85,B 0,C 180,E1 -16225.064,E2 -16225.064} C_VEL
LIN {X 0,Y 306.942,Z 617.556,A -85,B 0,C 180,E1 -16227.255,E2 -16227.255} C_VEL
LIN {X 0,Y 306.651,Z 614.021,A -85,B 0,C 180,E1 -16230.279,E2 -16230.279} C_VEL
LIN {X 0,Y 306.371,Z 611.124,A -85,B 0,C 180,E1 -16233.405,E2 -16233.405} C_VEL
LIN {X 0,Y 306.168,Z 608.96,A -85,B 0,C 180,E1 -16236.643,E2 -16236.643} C_VEL
LIN {X 0,Y 306.147,Z 607.763,A -85,B 0,C 180,E1 -16240,E2 -16240} C_VEL
LIN {X 0,Y 305.885,Z 607.924,A -85,B 0,C 180,E1 -16241.783,E2 -16241.783} C_VEL
LIN {X 0,Y 305.226,Z 609.045,A -85,B 0,C 180,E1 -16244.458,E2 -16244.458} C_VEL
LIN {X 0,Y 304.95,Z 610.522,A -85,B 0,C 180,E1 -16246.262,E2 -16246.262} C_VEL
LIN {X 0,Y 304.959,Z 614.877,A -85,B 0,C 180,E1 -16249.815,E2 -16249.815} C_VEL
LIN {X 0,Y 304.819,Z 618.306,A -85,B 0,C 180,E1 -16251.621,E2 -16251.621} C_VEL
LIN {X 0,Y 304.019,Z 625.303,A -85,B 0,C 180,E1 -16254.241,E2 -16254.241} C_VEL
LIN {X 0,Y 303.598,Z 634.927,A -85,B 0,C 180,E1 -16257.143,E2 -16257.143} C_VEL
LIN {X 0,Y 303.719,Z 645.075,A -85,B 0,C 180,E1 -16259.67,E2 -16259.67} C_VEL
LIN {X 0,Y 304.101,Z 653.821,A -85,B 0,C 180,E1 -16261.485,E2 -16261.485} C_VEL
LIN {X 0,Y 307.571,Z 667.034,A -85,B 0,C 180,E1 -16262.855,E2 -16262.855} C_VEL
LIN {X 0,Y 309.577,Z 679.317,A -85,B 0,C 180,E1 -16264.051,E2 -16264.051} C_VEL
LIN {X 0,Y 310.082,Z 689.635,A -85,B 0,C 180,E1 -16265.04,E2 -16265.04} C_VEL
LIN {X 0,Y 309.42,Z 701.329,A -85,B 0,C 180,E1 -16266.225,E2 -16266.225} C_VEL
LIN {X 0,Y 308.093,Z 713.791,A -85,B 0,C 180,E1 -16267.715,E2 -16267.715} C_VEL
LIN {X 0,Y 306.911,Z 720.941,A -85,B 0,C 180,E1 -16268.685,E2 -16268.685} C_VEL
LIN {X 0,Y 304.395,Z 732.11,A -85,B 0,C 180,E1 -16270.442,E2 -16270.442} C_VEL
LIN {X 0,Y 302.186,Z 741.985,A -85,B 0,C 180,E1 -16272.403,E2 -16272.403} C_VEL
LIN {X 0,Y 300.629,Z 748.889,A -85,B 0,C 180,E1 -16274.058,E2 -16274.058} C_VEL
LIN {X 0,Y 299.003,Z 756.813,A -85,B 0,C 180,E1 -16276.407,E2 -16276.407} C_VEL
LIN {X 0,Y 297.885,Z 762.216,A -85,B 0,C 180,E1 -16278.433,E2 -16278.433} C_VEL
LIN {X 0,Y 297.252,Z 766.5,A -85,B 0,C 180,E1 -16280.475,E2 -16280.475} C_VEL
LIN {X 0,Y 296.975,Z 768.763,A -85,B 0,C 180,E1 -16281.838,E2 -16281.838} C_VEL
LIN {X 0,Y 296.745,Z 771.582,A -85,B 0,C 180,E1 -16284.111,E2 -16284.111} C_VEL
LIN {X 0,Y 296.734,Z 773.017,A -85,B 0,C 180,E1 -16285.927,E2 -16285.927} C_VEL
LIN {X 0,Y 296.888,Z 773.721,A -85,B 0,C 180,E1 -16288.645,E2 -16288.645} C_VEL
LIN {X 0,Y 297.065,Z 773.465,A -85,B 0,C 180,E1 -16290.001,E2 -16290.001} C_VEL
LIN {X 0,Y 297.004,Z 772.732,A -85,B 0,C 180,E1 -16291.357,E2 -16291.357} C_VEL
LIN {X 0,Y 296.837,Z 771.541,A -85,B 0,C 180,E1 -16292.715,E2 -16292.715} C_VEL
LIN {X 0,Y 296.862,Z 768.935,A -85,B 0,C 180,E1 -16294.754,E2 -16294.754} C_VEL
LIN {X 0,Y 296.92,Z 765.231,A -85,B 0,C 180,E1 -16296.798,E2 -16296.798} C_VEL
LIN {X 0,Y 297.104,Z 760.33,A -85,B 0,C 180,E1 -16298.846,E2 -16298.846} C_VEL
LIN {X 0,Y 297.516,Z 754.108,A -85,B 0,C 180,E1 -16300.894,E2 -16300.894} C_VEL
LIN {X 0,Y 298.285,Z 746.287,A -85,B 0,C 180,E1 -16302.935,E2 -16302.935} C_VEL
LIN {X 0,Y 299.134,Z 738.305,A -85,B 0,C 180,E1 -16304.631,E2 -16304.631} C_VEL
LIN {X 0,Y 300.003,Z 729.626,A -85,B 0,C 180,E1 -16306.159,E2 -16306.159} C_VEL
LIN {X 0,Y 301.194,Z 719.25,A -85,B 0,C 180,E1 -16307.659,E2 -16307.659} C_VEL
LIN {X 0,Y 302.196,Z 709.274,A -85,B 0,C 180,E1 -16308.826,E2 -16308.826} C_VEL
LIN {X 0,Y 301.99,Z 696.188,A -85,B 0,C 180,E1 -16310.077,E2 -16310.077} C_VEL
LIN {X 0,Y 301.316,Z 683.082,A -85,B 0,C 180,E1 -16311.043,E2 -16311.043} C_VEL
LIN {X 0,Y 299.018,Z 656.841,A -85,B 0,C 180,E1 -16312.527,E2 -16312.527} C_VEL
LIN {X 0,Y 298.673,Z 653.637,A -85,B 0,C 180,E1 -16312.7,E2 -16312.7} C_VEL
LIN {X 0,Y 298.183,Z 645.576,A -85,B 0,C 180,E1 -16313.545,E2 -16313.545} C_VEL
LIN {X 0,Y 299.212,Z 633.977,A -85,B 0,C 180,E1 -16318.02,E2 -16318.02} C_VEL
LIN {X 0,Y 300.296,Z 624.315,A -85,B 0,C 180,E1 -16321.776,E2 -16321.776} C_VEL
LIN {X 0,Y 301.584,Z 614.568,A -85,B 0,C 180,E1 -16325.634,E2 -16325.634} C_VEL
LIN {X 0,Y 302.308,Z 609.23,A -85,B 0,C 180,E1 -16327.774,E2 -16327.774} C_VEL
LIN {X 0,Y 301.577,Z 603.565,A -85,B 0,C 180,E1 -16330.198,E2 -16330.198} C_VEL
LIN {X 0,Y 300.206,Z 596.311,A -85,B 0,C 180,E1 -16333.47,E2 -16333.47} C_VEL
LIN {X 0,Y 298.476,Z 587.686,A -85,B 0,C 180,E1 -16337.622,E2 -16337.622} C_VEL
LIN {X 0,Y 298.409,Z 587.315,A -85,B 0,C 180,E1 -16337.838,E2 -16337.838} C_VEL
LIN {X 0,Y 298.437,Z 587.315,A -85,B 0,C 180,E1 -16342.245,E2 -16342.245} C_VEL
LIN {X 0,Y 298.414,Z 587.314,A -85,B 0,C 180,E1 -16345.581,E2 -16345.581} C_VEL
LIN {X 0,Y 298.401,Z 587.315,A -85,B 0,C 180,E1 -16348.791,E2 -16348.791} C_VEL
LIN {X 0,Y 298.468,Z 587.306,A -85,B 0,C 180,E1 -16351.904,E2 -16351.904} C_VEL
LIN {X 0,Y 298.491,Z 587.302,A -85,B 0,C 180,E1 -16354.924,E2 -16354.924} C_VEL
LIN {X 0,Y 298.463,Z 587.305,A -85,B 0,C 180,E1 -16359.316,E2 -16359.316} C_VEL
LIN {X 0,Y 298.543,Z 587.299,A -85,B 0,C 180,E1 -16362.179,E2 -16362.179} C_VEL
LIN {X 0,Y 298.599,Z 587.289,A -85,B 0,C 180,E1 -16364.994,E2 -16364.994} C_VEL
LIN {X 0,Y 298.599,Z 587.288,A -85,B 0,C 180,E1 -16369.146,E2 -16369.146} C_VEL
LIN {X 0,Y 298.765,Z 587.268,A -85,B 0,C 180,E1 -16371.886,E2 -16371.886} C_VEL
LIN {X 0,Y 298.664,Z 587.283,A -85,B 0,C 180,E1 -16374.598,E2 -16374.598} C_VEL
LIN {X 0,Y 298.928,Z 587.249,A -85,B 0,C 180,E1 -16378.652,E2 -16378.652} C_VEL
LIN {X 0,Y 298.928,Z 587.245,A -85,B 0,C 180,E1 -16381.347,E2 -16381.347} C_VEL
LIN {X 0,Y 298.802,Z 587.263,A -85,B 0,C 180,E1 -16386.753,E2 -16386.753} C_VEL
LIN {X 0,Y 298.685,Z 587.276,A -85,B 0,C 180,E1 -16389.48,E2 -16389.48} C_VEL
LIN {X 0,Y 298.556,Z 587.291,A -85,B 0,C 180,E1 -16393.615,E2 -16393.615} C_VEL
LIN {X 0,Y 298.552,Z 587.293,A -85,B 0,C 180,E1 -16396.408,E2 -16396.408} C_VEL
LIN {X 0,Y 298.515,Z 587.297,A -85,B 0,C 180,E1 -16399.654,E2 -16399.654} C_VEL
LIN {X 0,Y 298.461,Z 587.304,A -85,B 0,C 180,E1 -16403.597,E2 -16403.597} C_VEL
LIN {X 0,Y 298.492,Z 587.301,A -85,B 0,C 180,E1 -16406.573,E2 -16406.573} C_VEL
LIN {X 0,Y 298.424,Z 587.308,A -85,B 0,C 180,E1 -16409.64,E2 -16409.64} C_VEL
LIN {X 0,Y 298.398,Z 587.314,A -85,B 0,C 180,E1 -16412.799,E2 -16412.799} C_VEL
LIN {X 0,Y 298.448,Z 587.308,A -85,B 0,C 180,E1 -16416.807,E2 -16416.807} C_VEL
LIN {X 0,Y 298.389,Z 587.314,A -85,B 0,C 180,E1 -16421.087,E2 -16421.087} C_VEL
LIN {X 0,Y 298.39,Z 587.311,A -85,B 0,C 180,E1 -16425.04,E2 -16425.04} C_VEL
LIN {X 0,Y 298.414,Z 587.313,A -85,B 0,C 180,E1 -16428.742,E2 -16428.742} C_VEL
LIN {X 0,Y 298.433,Z 587.309,A -85,B 0,C 180,E1 -16432.243,E2 -16432.243} C_VEL
LIN {X 0,Y 298.409,Z 587.311,A -85,B 0,C 180,E1 -16435.58,E2 -16435.58} C_VEL
LIN {X 0,Y 298.392,Z 587.316,A -85,B 0,C 180,E1 -16438.79,E2 -16438.79} C_VEL
LIN {X 0,Y 298.457,Z 587.306,A -85,B 0,C 180,E1 -16441.903,E2 -16441.903} C_VEL
LIN {X 0,Y 298.483,Z 587.304,A -85,B 0,C 180,E1 -16444.923,E2 -16444.923} C_VEL
LIN {X 0,Y 298.45,Z 587.306,A -85,B 0,C 180,E1 -16449.314,E2 -16449.314} C_VEL
LIN {X 0,Y 298.538,Z 587.298,A -85,B 0,C 180,E1 -16452.178,E2 -16452.178} C_VEL
LIN {X 0,Y 298.593,Z 587.29,A -85,B 0,C 180,E1 -16454.994,E2 -16454.994} C_VEL
LIN {X 0,Y 298.595,Z 587.29,A -85,B 0,C 180,E1 -16459.146,E2 -16459.146} C_VEL
LIN {X 0,Y 298.789,Z 587.269,A -85,B 0,C 180,E1 -16462.438,E2 -16462.438} C_VEL
LIN {X 0,Y 302.027,Z 598.013,A -85,B 0,C 180,E1 -16463.485,E2 -16463.485} C_VEL
LIN {X 0,Y 305.369,Z 609.865,A -85,B 0,C 180,E1 -16464.888,E2 -16464.888} C_VEL
LIN {X 0,Y 305.684,Z 611.557,A -85,B 0,C 180,E1 -16465.099,E2 -16465.099} C_VEL
LIN {X 0,Y 304.589,Z 622.871,A -85,B 0,C 180,E1 -16466.526,E2 -16466.526} C_VEL
LIN {X 0,Y 303.646,Z 632.289,A -85,B 0,C 180,E1 -16468.009,E2 -16468.009} C_VEL
LIN {X 0,Y 302.522,Z 641.008,A -85,B 0,C 180,E1 -16469.678,E2 -16469.678} C_VEL
LIN {X 0,Y 301.493,Z 649.353,A -85,B 0,C 180,E1 -16471.668,E2 -16471.668} C_VEL
LIN {X 0,Y 300.655,Z 656.105,A -85,B 0,C 180,E1 -16473.684,E2 -16473.684} C_VEL
LIN {X 0,Y 299.78,Z 662.358,A -85,B 0,C 180,E1 -16476.055,E2 -16476.055} C_VEL
LIN {X 0,Y 299.254,Z 666.441,A -85,B 0,C 180,E1 -16478.099,E2 -16478.099} C_VEL
LIN {X 0,Y 299.002,Z 668.563,A -85,B 0,C 180,E1 -16479.469,E2 -16479.469} C_VEL
LIN {X 0,Y 298.834,Z 670.256,A -85,B 0,C 180,E1 -16480.843,E2 -16480.843} C_VEL
LIN {X 0,Y 298.78,Z 671.544,A -85,B 0,C 180,E1 -16482.221,E2 -16482.221} C_VEL
LIN {X 0,Y 298.774,Z 672.414,A -85,B 0,C 180,E1 -16483.604,E2 -16483.604} C_VEL
LIN {X 0,Y 299.087,Z 672.908,A -85,B 0,C 180,E1 -16486.377,E2 -16486.377} C_VEL
LIN {X 0,Y 299.332,Z 672.576,A -85,B 0,C 180,E1 -16487.77,E2 -16487.77} C_VEL
LIN {X 0,Y 299.674,Z 671.786,A -85,B 0,C 180,E1 -16489.166,E2 -16489.166} C_VEL
LIN {X 0,Y 300.176,Z 670.573,A -85,B 0,C 180,E1 -16490.559,E2 -16490.559} C_VEL
LIN {X 0,Y 301.075,Z 667.932,A -85,B 0,C 180,E1 -16492.652,E2 -16492.652} C_VEL
LIN {X 0,Y 302.278,Z 663.819,A -85,B 0,C 180,E1 -16494.941,E2 -16494.941} C_VEL
LIN {X 0,Y 303.517,Z 659.272,A -85,B 0,C 180,E1 -16496.84,E2 -16496.84} C_VEL
LIN {X 0,Y 305.103,Z 652.943,A -85,B 0,C 180,E1 -16498.928,E2 -16498.928} C_VEL
LIN {X 0,Y 306.972,Z 644.851,A -85,B 0,C 180,E1 -16501.004,E2 -16501.004} C_VEL
LIN {X 0,Y 308.829,Z 635.957,A -85,B 0,C 180,E1 -16502.824,E2 -16502.824} C_VEL
LIN {X 0,Y 310.552,Z 626.022,A -85,B 0,C 180,E1 -16504.454,E2 -16504.454} C_VEL
LIN {X 0,Y 311.184,Z 621.982,A -85,B 0,C 180,E1 -16505.022,E2 -16505.022} C_VEL
LIN {X 0,Y 308.668,Z 612.572,A -85,B 0,C 180,E1 -16506.594,E2 -16506.594} C_VEL
LIN {X 0,Y 307.36,Z 608.666,A -85,B 0,C 180,E1 -16507.212,E2 -16507.212} C_VEL
LIN {X 0,Y 301.917,Z 600.784,A -85,B 0,C 180,E1 -16508.681,E2 -16508.681} C_VEL
LIN {X 0,Y 300.561,Z 598.783,A -85,B 0,C 180,E1 -16509.028,E2 -16509.028} C_VEL
LIN {X 0,Y 300.429,Z 598.29,A -85,B 0,C 180,E1 -16509.13,E2 -16509.13} C_VEL
LIN {X 0,Y 300.686,Z 603.349,A -85,B 0,C 180,E1 -16511.588,E2 -16511.588} C_VEL
LIN {X 0,Y 300.24,Z 611.445,A -85,B 0,C 180,E1 -16515.394,E2 -16515.394} C_VEL
LIN {X 0,Y 299.739,Z 619.105,A -85,B 0,C 180,E1 -16518.966,E2 -16518.966} C_VEL
LIN {X 0,Y 299.33,Z 627.679,A -85,B 0,C 180,E1 -16522.964,E2 -16522.964} C_VEL
LIN {X 0,Y 299.15,Z 631.876,A -85,B 0,C 180,E1 -16524.909,E2 -16524.909} C_VEL
LIN {X 0,Y 301.721,Z 646.298,A -85,B 0,C 180,E1 -16525.765,E2 -16525.765} C_VEL
LIN {X 0,Y 303.969,Z 659.45,A -85,B 0,C 180,E1 -16526.803,E2 -16526.803} C_VEL
LIN {X 0,Y 304.276,Z 662.671,A -85,B 0,C 180,E1 -16527.093,E2 -16527.093} C_VEL
LIN {X 0,Y 303.313,Z 674.217,A -85,B 0,C 180,E1 -16528.189,E2 -16528.189} C_VEL
LIN {X 0,Y 302.036,Z 685.974,A -85,B 0,C 180,E1 -16529.597,E2 -16529.597} C_VEL
LIN {X 0,Y 300.847,Z 696.698,A -85,B 0,C 180,E1 -16531.197,E2 -16531.197} C_VEL
LIN {X 0,Y 299.776,Z 706.37,A -85,B 0,C 180,E1 -16532.98,E2 -16532.98} C_VEL
LIN {X 0,Y 298.721,Z 715.041,A -85,B 0,C 180,E1 -16534.946,E2 -16534.946} C_VEL
LIN {X 0,Y 298.026,Z 721.96,A -85,B 0,C 180,E1 -16536.877,E2 -16536.877} C_VEL
LIN {X 0,Y 297.36,Z 728.629,A -85,B 0,C 180,E1 -16539.237,E2 -16539.237} C_VEL
LIN {X 0,Y 296.993,Z 732.9,A -85,B 0,C 180,E1 -16541.178,E2 -16541.178} C_VEL
LIN {X 0,Y 296.663,Z 736.71,A -85,B 0,C 180,E1 -16543.505,E2 -16543.505} C_VEL
LIN {X 0,Y 295.914,Z 738.093,A -85,B 0,C 180,E1 -16544.612,E2 -16544.612} C_VEL
LIN {X 0,Y 293.014,Z 739.816,A -85,B 0,C 180,E1 -16546.429,E2 -16546.429} C_VEL
LIN {X 0,Y 290.663,Z 740.741,A -85,B 0,C 180,E1 -16547.914,E2 -16547.914} C_VEL
LIN {X 0,Y 289.701,Z 741.153,A -85,B 0,C 180,E1 -16549.267,E2 -16549.267} C_VEL
LIN {X 0,Y 289.705,Z 741.099,A -85,B 0,C 180,E1 -16549.462,E2 -16549.462} C_VEL
LIN {X 0,Y 290.089,Z 740.809,A -85,B 0,C 180,E1 -16551.642,E2 -16551.642} C_VEL
LIN {X 0,Y 290.471,Z 740.036,A -85,B 0,C 180,E1 -16553.052,E2 -16553.052} C_VEL
LIN {X 0,Y 290.884,Z 738.88,A -85,B 0,C 180,E1 -16554.455,E2 -16554.455} C_VEL
LIN {X 0,Y 291.672,Z 736.346,A -85,B 0,C 180,E1 -16556.547,E2 -16556.547} C_VEL
LIN {X 0,Y 292.804,Z 732.799,A -85,B 0,C 180,E1 -16558.625,E2 -16558.625} C_VEL
LIN {X 0,Y 294.167,Z 728.201,A -85,B 0,C 180,E1 -16560.685,E2 -16560.685} C_VEL
LIN {X 0,Y 295.895,Z 722.429,A -85,B 0,C 180,E1 -16562.723,E2 -16562.723} C_VEL
LIN {X 0,Y 297.948,Z 715.242,A -85,B 0,C 180,E1 -16564.736,E2 -16564.736} C_VEL
LIN {X 0,Y 300.352,Z 706.384,A -85,B 0,C 180,E1 -16566.719,E2 -16566.719} C_VEL
LIN {X 0,Y 302.807,Z 696.516,A -85,B 0,C 180,E1 -16568.509,E2 -16568.509} C_VEL
LIN {X 0,Y 305.315,Z 685.438,A -85,B 0,C 180,E1 -16570.109,E2 -16570.109} C_VEL
LIN {X 0,Y 307.454,Z 674.51,A -85,B 0,C 180,E1 -16571.371,E2 -16571.371} C_VEL
LIN {X 0,Y 306.66,Z 666.669,A -85,B 0,C 180,E1 -16572.462,E2 -16572.462} C_VEL
LIN {X 0,Y 304.213,Z 655.902,A -85,B 0,C 180,E1 -16574.007,E2 -16574.007} C_VEL
LIN {X 0,Y 300.521,Z 645.125,A -85,B 0,C 180,E1 -16575.623,E2 -16575.623} C_VEL
LIN {X 0,Y 297.591,Z 638.1,A -85,B 0,C 180,E1 -16576.728,E2 -16576.728} C_VEL
LIN {X 0,Y 298.957,Z 631.197,A -85,B 0,C 180,E1 -16580.649,E2 -16580.649} C_VEL
LIN {X 0,Y 300.259,Z 625.434,A -85,B 0,C 180,E1 -16584.102,E2 -16584.102} C_VEL
LIN {X 0,Y 300.694,Z 622.134,A -85,B 0,C 180,E1 -16586.365,E2 -16586.365} C_VEL
LIN {X 0,Y 300.6,Z 618.499,A -85,B 0,C 180,E1 -16589.405,E2 -16589.405} C_VEL
LIN {X 0,Y 300.369,Z 615.537,A -85,B 0,C 180,E1 -16592.617,E2 -16592.617} C_VEL
LIN {X 0,Y 300.195,Z 613.328,A -85,B 0,C 180,E1 -16595.824,E2 -16595.824} C_VEL
LIN {X 0,Y 300.215,Z 612.509,A -85,B 0,C 180,E1 -16597.493,E2 -16597.493} C_VEL
LIN {X 0,Y 300.297,Z 611.972,A -85,B 0,C 180,E1 -16599.44,E2 -16599.44} C_VEL
LIN {X 0,Y 300.219,Z 612.081,A -85,B 0,C 180,E1 -16601.489,E2 -16601.489} C_VEL
LIN {X 0,Y 299.869,Z 612.929,A -85,B 0,C 180,E1 -16603.405,E2 -16603.405} C_VEL
LIN {X 0,Y 299.428,Z 614.09,A -85,B 0,C 180,E1 -16605.242,E2 -16605.242} C_VEL
LIN {X 0,Y 299.261,Z 617.981,A -85,B 0,C 180,E1 -16608.722,E2 -16608.722} C_VEL
LIN {X 0,Y 299.428,Z 619.871,A -85,B 0,C 180,E1 -16610.006,E2 -16610.006} C_VEL
LIN {X 0,Y 299.068,Z 623.903,A -85,B 0,C 180,E1 -16611.896,E2 -16611.896} C_VEL
LIN {X 0,Y 298.396,Z 629.434,A -85,B 0,C 180,E1 -16613.929,E2 -16613.929} C_VEL
LIN {X 0,Y 297.896,Z 639.986,A -85,B 0,C 180,E1 -16617.14,E2 -16617.14} C_VEL
LIN {X 0,Y 297.876,Z 650.12,A -85,B 0,C 180,E1 -16619.622,E2 -16619.622} C_VEL
LIN {X 0,Y 298.063,Z 653.442,A -85,B 0,C 180,E1 -16620.322,E2 -16620.322} C_VEL
LIN {X 0,Y 301.58,Z 666.742,A -85,B 0,C 180,E1 -16621.842,E2 -16621.842} C_VEL
LIN {X 0,Y 303.392,Z 677.33,A -85,B 0,C 180,E1 -16622.942,E2 -16622.942} C_VEL
LIN {X 0,Y 304.17,Z 687.052,A -85,B 0,C 180,E1 -16623.961,E2 -16623.961} C_VEL
LIN {X 0,Y 303.688,Z 698.636,A -85,B 0,C 180,E1 -16625.162,E2 -16625.162} C_VEL
LIN {X 0,Y 302.338,Z 710.437,A -85,B 0,C 180,E1 -16626.543,E2 -16626.543} C_VEL
LIN {X 0,Y 301.154,Z 718.877,A -85,B 0,C 180,E1 -16627.716,E2 -16627.716} C_VEL
LIN {X 0,Y 298.729,Z 729.308,A -85,B 0,C 180,E1 -16629.337,E2 -16629.337} C_VEL
LIN {X 0,Y 296.574,Z 738.052,A -85,B 0,C 180,E1 -16630.985,E2 -16630.985} C_VEL
LIN {X 0,Y 294.506,Z 746.183,A -85,B 0,C 180,E1 -16632.848,E2 -16632.848} C_VEL
LIN {X 0,Y 292.804,Z 753.919,A -85,B 0,C 180,E1 -16635.048,E2 -16635.048} C_VEL
LIN {X 0,Y 291.187,Z 760.627,A -85,B 0,C 180,E1 -16637.456,E2 -16637.456} C_VEL
LIN {X 0,Y 290.414,Z 765.135,A -85,B 0,C 180,E1 -16639.544,E2 -16639.544} C_VEL
LIN {X 0,Y 289.913,Z 768.598,A -85,B 0,C 180,E1 -16641.638,E2 -16641.638} C_VEL
LIN {X 0,Y 289.639,Z 771.524,A -85,B 0,C 180,E1 -16644.188,E2 -16644.188} C_VEL
LIN {X 0,Y 289.644,Z 772.652,A -85,B 0,C 180,E1 -16645.827,E2 -16645.827} C_VEL
LIN {X 0,Y 289.666,Z 773.156,A -85,B 0,C 180,E1 -16647.22,E2 -16647.22} C_VEL
LIN {X 0,Y 289.795,Z 773.261,A -85,B 0,C 180,E1 -16648.612,E2 -16648.612} C_VEL
LIN {X 0,Y 290.005,Z 772.938,A -85,B 0,C 180,E1 -16650.001,E2 -16650.001} C_VEL
LIN {X 0,Y 289.927,Z 772.136,A -85,B 0,C 180,E1 -16651.39,E2 -16651.39} C_VEL
LIN {X 0,Y 289.753,Z 770.904,A -85,B 0,C 180,E1 -16652.782,E2 -16652.782} C_VEL
LIN {X 0,Y 289.806,Z 768.216,A -85,B 0,C 180,E1 -16654.87,E2 -16654.87} C_VEL
LIN {X 0,Y 289.855,Z 764.406,A -85,B 0,C 180,E1 -16656.964,E2 -16656.964} C_VEL
LIN {X 0,Y 290.047,Z 759.393,A -85,B 0,C 180,E1 -16659.063,E2 -16659.063} C_VEL
LIN {X 0,Y 290.496,Z 753.011,A -85,B 0,C 180,E1 -16661.161,E2 -16661.161} C_VEL
LIN {X 0,Y 291.291,Z 745.02,A -85,B 0,C 180,E1 -16663.252,E2 -16663.252} C_VEL
LIN {X 0,Y 292.234,Z 736.889,A -85,B 0,C 180,E1 -16664.984,E2 -16664.984} C_VEL
LIN {X 0,Y 293.137,Z 728.089,A -85,B 0,C 180,E1 -16666.538,E2 -16666.538} C_VEL
LIN {X 0,Y 294.36,Z 717.301,A -85,B 0,C 180,E1 -16668.083,E2 -16668.083} C_VEL
LIN {X 0,Y 295.178,Z 708.612,A -85,B 0,C 180,E1 -16669.111,E2 -16669.111} C_VEL
LIN {X 0,Y 294.965,Z 695.489,A -85,B 0,C 180,E1 -16670.395,E2 -16670.395} C_VEL
LIN {X 0,Y 294.286,Z 682.14,A -85,B 0,C 180,E1 -16671.395,E2 -16671.395} C_VEL
LIN {X 0,Y 292.166,Z 657.431,A -85,B 0,C 180,E1 -16672.89,E2 -16672.89} C_VEL
LIN {X 0,Y 291.666,Z 653.044,A -85,B 0,C 180,E1 -16673.117,E2 -16673.117} C_VEL
LIN {X 0,Y 291.181,Z 644.359,A -85,B 0,C 180,E1 -16674.113,E2 -16674.113} C_VEL
LIN {X 0,Y 292.321,Z 632.671,A -85,B 0,C 180,E1 -16678.742,E2 -16678.742} C_VEL
LIN {X 0,Y 293.741,Z 621.08,A -85,B 0,C 180,E1 -16683.388,E2 -16683.388} C_VEL
LIN {X 0,Y 295.155,Z 611.312,A -85,B 0,C 180,E1 -16687.387,E2 -16687.387} C_VEL
LIN {X 0,Y 295.167,Z 608.244,A -85,B 0,C 180,E1 -16688.684,E2 -16688.684} C_VEL
LIN {X 0,Y 293.819,Z 600.59,A -85,B 0,C 180,E1 -16692.139,E2 -16692.139} C_VEL
LIN {X 0,Y 292.157,Z 592.155,A -85,B 0,C 180,E1 -16696.194,E2 -16696.194} C_VEL
LIN {X 0,Y 291.361,Z 588.194,A -85,B 0,C 180,E1 -16698.267,E2 -16698.267} C_VEL
LIN {X 0,Y 291.37,Z 588.192,A -85,B 0,C 180,E1 -16701.16,E2 -16701.16} C_VEL
LIN {X 0,Y 291.391,Z 588.191,A -85,B 0,C 180,E1 -16704.63,E2 -16704.63} C_VEL
LIN {X 0,Y 291.378,Z 588.192,A -85,B 0,C 180,E1 -16707.951,E2 -16707.951} C_VEL
LIN {X 0,Y 291.387,Z 588.187,A -85,B 0,C 180,E1 -16711.158,E2 -16711.158} C_VEL
LIN {X 0,Y 291.42,Z 588.187,A -85,B 0,C 180,E1 -16714.272,E2 -16714.272} C_VEL
LIN {X 0,Y 291.394,Z 588.185,A -85,B 0,C 180,E1 -16717.3,E2 -16717.3} C_VEL
LIN {X 0,Y 291.464,Z 588.182,A -85,B 0,C 180,E1 -16720.27,E2 -16720.27} C_VEL
LIN {X 0,Y 291.561,Z 588.168,A -85,B 0,C 180,E1 -16724.623,E2 -16724.623} C_VEL
LIN {X 0,Y 291.542,Z 588.168,A -85,B 0,C 180,E1 -16728.88,E2 -16728.88} C_VEL
LIN {X 0,Y 291.716,Z 588.145,A -85,B 0,C 180,E1 -16731.688,E2 -16731.688} C_VEL
LIN {X 0,Y 291.635,Z 588.159,A -85,B 0,C 180,E1 -16734.468,E2 -16734.468} C_VEL
LIN {X 0,Y 291.894,Z 588.126,A -85,B 0,C 180,E1 -16738.62,E2 -16738.62} C_VEL
LIN {X 0,Y 291.894,Z 588.121,A -85,B 0,C 180,E1 -16741.379,E2 -16741.379} C_VEL
LIN {X 0,Y 291.751,Z 588.14,A -85,B 0,C 180,E1 -16746.917,E2 -16746.917} C_VEL
LIN {X 0,Y 291.634,Z 588.155,A -85,B 0,C 180,E1 -16749.711,E2 -16749.711} C_VEL
LIN {X 0,Y 291.526,Z 588.168,A -85,B 0,C 180,E1 -16753.95,E2 -16753.95} C_VEL
LIN {X 0,Y 291.491,Z 588.171,A -85,B 0,C 180,E1 -16756.817,E2 -16756.817} C_VEL
LIN {X 0,Y 291.454,Z 588.177,A -85,B 0,C 180,E1 -16759.874,E2 -16759.874} C_VEL
LIN {X 0,Y 291.404,Z 588.186,A -85,B 0,C 180,E1 -16764.204,E2 -16764.204} C_VEL
LIN {X 0,Y 291.426,Z 588.177,A -85,B 0,C 180,E1 -16767.271,E2 -16767.271} C_VEL
LIN {X 0,Y 291.34,Z 588.196,A -85,B 0,C 180,E1 -16770.436,E2 -16770.436} C_VEL
LIN {X 0,Y 291.347,Z 588.19,A -85,B 0,C 180,E1 -16773.697,E2 -16773.697} C_VEL
LIN {X 0,Y 291.378,Z 588.187,A -85,B 0,C 180,E1 -16777.253,E2 -16777.253} C_VEL
LIN {X 0,Y 291.335,Z 588.196,A -85,B 0,C 180,E1 -16780.641,E2 -16780.641} C_VEL
LIN {X 0,Y 291.316,Z 588.196,A -85,B 0,C 180,E1 -16784.396,E2 -16784.396} C_VEL
LIN {X 0,Y 291.352,Z 588.194,A -85,B 0,C 180,E1 -16788.398,E2 -16788.398} C_VEL
LIN {X 0,Y 291.366,Z 588.186,A -85,B 0,C 180,E1 -16791.159,E2 -16791.159} C_VEL
LIN {X 0,Y 291.386,Z 588.19,A -85,B 0,C 180,E1 -16794.628,E2 -16794.628} C_VEL
LIN {X 0,Y 291.371,Z 588.187,A -85,B 0,C 180,E1 -16797.949,E2 -16797.949} C_VEL
LIN {X 0,Y 291.377,Z 588.188,A -85,B 0,C 180,E1 -16801.157,E2 -16801.157} C_VEL
LIN {X 0,Y 291.413,Z 588.184,A -85,B 0,C 180,E1 -16804.27,E2 -16804.27} C_VEL
LIN {X 0,Y 291.382,Z 588.186,A -85,B 0,C 180,E1 -16807.298,E2 -16807.298} C_VEL
LIN {X 0,Y 291.458,Z 588.18,A -85,B 0,C 180,E1 -16810.269,E2 -16810.269} C_VEL
LIN {X 0,Y 291.555,Z 588.166,A -85,B 0,C 180,E1 -16814.622,E2 -16814.622} C_VEL
LIN {X 0,Y 291.538,Z 588.17,A -85,B 0,C 180,E1 -16818.879,E2 -16818.879} C_VEL
LIN {X 0,Y 291.741,Z 588.144,A -85,B 0,C 180,E1 -16821.993,E2 -16821.993} C_VEL
LIN {X 0,Y 295.299,Z 599.687,A -85,B 0,C 180,E1 -16823.165,E2 -16823.165} C_VEL
LIN {X 0,Y 298.52,Z 611.386,A -85,B 0,C 180,E1 -16824.595,E2 -16824.595} C_VEL
LIN {X 0,Y 298.823,Z 612.749,A -85,B 0,C 180,E1 -16824.776,E2 -16824.776} C_VEL
LIN {X 0,Y 297.724,Z 624.286,A -85,B 0,C 180,E1 -16826.277,E2 -16826.277} C_VEL
LIN {X 0,Y 296.62,Z 634.601,A -85,B 0,C 180,E1 -16827.962,E2 -16827.962} C_VEL
LIN {X 0,Y 295.496,Z 642.895,A -85,B 0,C 180,E1 -16829.631,E2 -16829.631} C_VEL
LIN {X 0,Y 294.452,Z 651.185,A -85,B 0,C 180,E1 -16831.708,E2 -16831.708} C_VEL
LIN {X 0,Y 293.574,Z 657.798,A -85,B 0,C 180,E1 -16833.773,E2 -16833.773} C_VEL
LIN {X 0,Y 292.699,Z 663.877,A -85,B 0,C 180,E1 -16836.202,E2 -16836.202} C_VEL
LIN {X 0,Y 292.187,Z 667.836,A -85,B 0,C 180,E1 -16838.296,E2 -16838.296} C_VEL
LIN {X 0,Y 291.925,Z 669.89,A -85,B 0,C 180,E1 -16839.701,E2 -16839.701} C_VEL
LIN {X 0,Y 291.803,Z 671.524,A -85,B 0,C 180,E1 -16841.108,E2 -16841.108} C_VEL
LIN {X 0,Y 291.735,Z 672.746,A -85,B 0,C 180,E1 -16842.521,E2 -16842.521} C_VEL
LIN {X 0,Y 291.935,Z 673.907,A -85,B 0,C 180,E1 -16845.354,E2 -16845.354} C_VEL
LIN {X 0,Y 292.122,Z 673.915,A -85,B 0,C 180,E1 -16846.779,E2 -16846.779} C_VEL
LIN {X 0,Y 292.43,Z 673.48,A -85,B 0,C 180,E1 -16848.204,E2 -16848.204} C_VEL
LIN {X 0,Y 293.257,Z 671.583,A -85,B 0,C 180,E1 -16850.831,E2 -16850.831} C_VEL
LIN {X 0,Y 294.325,Z 668.602,A -85,B 0,C 180,E1 -16853.202,E2 -16853.202} C_VEL
LIN {X 0,Y 295.539,Z 664.719,A -85,B 0,C 180,E1 -16855.359,E2 -16855.359} C_VEL
LIN {X 0,Y 297.239,Z 658.663,A -85,B 0,C 180,E1 -16857.836,E2 -16857.836} C_VEL
LIN {X 0,Y 299.011,Z 651.878,A -85,B 0,C 180,E1 -16859.963,E2 -16859.963} C_VEL
LIN {X 0,Y 300.673,Z 644.855,A -85,B 0,C 180,E1 -16861.729,E2 -16861.729} C_VEL
LIN {X 0,Y 302.672,Z 635.599,A -85,B 0,C 180,E1 -16863.599,E2 -16863.599} C_VEL
LIN {X 0,Y 304.439,Z 625.426,A -85,B 0,C 180,E1 -16865.247,E2 -16865.247} C_VEL
LIN {X 0,Y 304.593,Z 623.488,A -85,B 0,C 180,E1 -16865.546,E2 -16865.546} C_VEL
LIN {X 0,Y 301.919,Z 613.73,A -85,B 0,C 180,E1 -16867.243,E2 -16867.243} C_VEL
LIN {X 0,Y 300.275,Z 610.692,A -85,B 0,C 180,E1 -16867.822,E2 -16867.822} C_VEL
LIN {X 0,Y 293.754,Z 601.505,A -85,B 0,C 180,E1 -16869.64,E2 -16869.64} C_VEL
LIN {X 0,Y 293.604,Z 600.995,A -85,B 0,C 180,E1 -16869.739,E2 -16869.739} C_VEL
LIN {X 0,Y 293.661,Z 605.87,A -85,B 0,C 180,E1 -16872.107,E2 -16872.107} C_VEL
LIN {X 0,Y 293.182,Z 613.994,A -85,B 0,C 180,E1 -16875.982,E2 -16875.982} C_VEL
LIN {X 0,Y 292.544,Z 624.169,A -85,B 0,C 180,E1 -16880.784,E2 -16880.784} C_VEL
LIN {X 0,Y 292.16,Z 632.227,A -85,B 0,C 180,E1 -16884.557,E2 -16884.557} C_VEL
LIN {X 0,Y 294.603,Z 645.902,A -85,B 0,C 180,E1 -16885.385,E2 -16885.385} C_VEL
LIN {X 0,Y 296.984,Z 660.047,A -85,B 0,C 180,E1 -16886.527,E2 -16886.527} C_VEL
LIN {X 0,Y 297.278,Z 663.789,A -85,B 0,C 180,E1 -16886.873,E2 -16886.873} C_VEL
LIN {X 0,Y 296.157,Z 676.383,A -85,B 0,C 180,E1 -16888.13,E2 -16888.13} C_VEL
LIN {X 0,Y 294.836,Z 688.238,A -85,B 0,C 180,E1 -16889.634,E2 -16889.634} C_VEL
LIN {X 0,Y 293.699,Z 698.269,A -85,B 0,C 180,E1 -16891.212,E2 -16891.212} C_VEL
LIN {X 0,Y 292.503,Z 708.594,A -85,B 0,C 180,E1 -16893.224,E2 -16893.224} C_VEL
LIN {X 0,Y 291.577,Z 716.232,A -85,B 0,C 180,E1 -16895.052,E2 -16895.052} C_VEL
LIN {X 0,Y 290.82,Z 723.639,A -85,B 0,C 180,E1 -16897.254,E2 -16897.254} C_VEL
LIN {X 0,Y 290.211,Z 729.493,A -85,B 0,C 180,E1 -16899.443,E2 -16899.443} C_VEL
LIN {X 0,Y 289.842,Z 734.026,A -85,B 0,C 180,E1 -16901.626,E2 -16901.626} C_VEL
LIN {X 0,Y 289.583,Z 736.881,A -85,B 0,C 180,E1 -16903.471,E2 -16903.471} C_VEL
LIN {X 0,Y 289.521,Z 739.627,A -85,B 0,C 180,E1 -16905.952,E2 -16905.952} C_VEL
LIN {X 0,Y 289.565,Z 740.556,A -85,B 0,C 180,E1 -16907.383,E2 -16907.383} C_VEL
LIN {X 0,Y 289.705,Z 741.099,A -85,B 0,C 180,E1 -16909.462,E2 -16909.462} C_VEL
LIN {X 0,Y 289.224,Z 741.142,A -85,B 0,C 180,E1 -16910.627,E2 -16910.627} C_VEL
LIN {X 0,Y 286.774,Z 740.715,A -85,B 0,C 180,E1 -16912.535,E2 -16912.535} C_VEL
LIN {X 0,Y 284.79,Z 739.955,A -85,B 0,C 180,E1 -16914.076,E2 -16914.076} C_VEL
LIN {X 0,Y 284.15,Z 739.005,A -85,B 0,C 180,E1 -16915.25,E2 -16915.25} C_VEL
LIN {X 0,Y 284.213,Z 738.56,A -85,B 0,C 180,E1 -16915.642,E2 -16915.642} C_VEL
LIN {X 0,Y 285.271,Z 735.551,A -85,B 0,C 180,E1 -16917.883,E2 -16917.883} C_VEL
LIN {X 0,Y 286.626,Z 731.625,A -85,B 0,C 180,E1 -16920.001,E2 -16920.001} C_VEL
LIN {X 0,Y 288.343,Z 726.422,A -85,B 0,C 180,E1 -16922.155,E2 -16922.155} C_VEL
LIN {X 0,Y 290.628,Z 719.108,A -85,B 0,C 180,E1 -16924.508,E2 -16924.508} C_VEL
LIN {X 0,Y 293.006,Z 711.144,A -85,B 0,C 180,E1 -16926.543,E2 -16926.543} C_VEL
LIN {X 0,Y 295.336,Z 703.061,A -85,B 0,C 180,E1 -16928.209,E2 -16928.209} C_VEL
LIN {X 0,Y 297.813,Z 693.36,A -85,B 0,C 180,E1 -16929.852,E2 -16929.852} C_VEL
LIN {X 0,Y 300.537,Z 681.488,A -85,B 0,C 180,E1 -16931.466,E2 -16931.466} C_VEL
LIN {X 0,Y 301.629,Z 675.972,A -85,B 0,C 180,E1 -16932.105,E2 -16932.105} C_VEL
LIN {X 0,Y 300.79,Z 668.401,A -85,B 0,C 180,E1 -16933.238,E2 -16933.238} C_VEL
LIN {X 0,Y 298.921,Z 659.317,A -85,B 0,C 180,E1 -16934.627,E2 -16934.627} C_VEL
LIN {X 0,Y 295.536,Z 648.921,A -85,B 0,C 180,E1 -16936.311,E2 -16936.311} C_VEL
LIN {X 0,Y 292.676,Z 641.87,A -85,B 0,C 180,E1 -16937.538,E2 -16937.538} C_VEL
LIN {X 0,Y 291.476,Z 638.714,A -85,B 0,C 180,E1 -16938.068,E2 -16938.068} C_VEL
LIN {X 0,Y 293.225,Z 631.237,A -85,B 0,C 180,E1 -16942.55,E2 -16942.55} C_VEL
LIN {X 0,Y 294.27,Z 626.782,A -85,B 0,C 180,E1 -16945.461,E2 -16945.461} C_VEL
LIN {X 0,Y 294.467,Z 623.655,A -85,B 0,C 180,E1 -16947.988,E2 -16947.988} C_VEL
LIN {X 0,Y 294.344,Z 620.857,A -85,B 0,C 180,E1 -16950.736,E2 -16950.736} C_VEL
LIN {X 0,Y 294.29,Z 618.768,A -85,B 0,C 180,E1 -16953.317,E2 -16953.317} C_VEL
LIN {X 0,Y 294.331,Z 616.939,A -85,B 0,C 180,E1 -16956.652,E2 -16956.652} C_VEL
LIN {X 0,Y 294.464,Z 616.379,A -85,B 0,C 180,E1 -16958.356,E2 -16958.356} C_VEL
LIN {X 0,Y 294.549,Z 616.177,A -85,B 0,C 180,E1 -16960.226,E2 -16960.226} C_VEL
LIN {X 0,Y 294.344,Z 616.646,A -85,B 0,C 180,E1 -16962.256,E2 -16962.256} C_VEL
LIN {X 0,Y 294.036,Z 617.765,A -85,B 0,C 180,E1 -16964.19,E2 -16964.19} C_VEL
LIN {X 0,Y 293.729,Z 620.678,A -85,B 0,C 180,E1 -16967.174,E2 -16967.174} C_VEL
LIN {X 0,Y 293.921,Z 624.5,A -85,B 0,C 180,E1 -16969.922,E2 -16969.922} C_VEL
LIN {X 0,Y 293.535,Z 627.856,A -85,B 0,C 180,E1 -16971.503,E2 -16971.503} C_VEL
LIN {X 0,Y 292.652,Z 634.607,A -85,B 0,C 180,E1 -16973.961,E2 -16973.961} C_VEL
LIN {X 0,Y 292.097,Z 644.279,A -85,B 0,C 180,E1 -16976.903,E2 -16976.903} C_VEL
LIN {X 0,Y 292.056,Z 652.707,A -85,B 0,C 180,E1 -16979.004,E2 -16979.004} C_VEL
LIN {X 0,Y 295.776,Z 666.944,A -85,B 0,C 180,E1 -16980.777,E2 -16980.777} C_VEL
LIN {X 0,Y 297.569,Z 677.324,A -85,B 0,C 180,E1 -16981.973,E2 -16981.973} C_VEL
LIN {X 0,Y 298.403,Z 688.998,A -85,B 0,C 180,E1 -16983.272,E2 -16983.272} C_VEL
LIN {X 0,Y 297.578,Z 701.153,A -85,B 0,C 180,E1 -16984.623,E2 -16984.623} C_VEL
LIN {X 0,Y 295.665,Z 714.672,A -85,B 0,C 180,E1 -16986.353,E2 -16986.353} C_VEL
LIN {X 0,Y 294.438,Z 721.44,A -85,B 0,C 180,E1 -16987.365,E2 -16987.365} C_VEL
LIN {X 0,Y 291.695,Z 732.223,A -85,B 0,C 180,E1 -16989.185,E2 -16989.185} C_VEL
LIN {X 0,Y 289.5,Z 740.339,A -85,B 0,C 180,E1 -16990.87,E2 -16990.87} C_VEL
LIN {X 0,Y 287.276,Z 748.535,A -85,B 0,C 180,E1 -16992.93,E2 -16992.93} C_VEL
LIN {X 0,Y 285.727,Z 755.259,A -85,B 0,C 180,E1 -16995.034,E2 -16995.034} C_VEL
LIN {X 0,Y 284.235,Z 760.741,A -85,B 0,C 180,E1 -16997.144,E2 -16997.144} C_VEL
LIN {X 0,Y 283.399,Z 765.118,A -85,B 0,C 180,E1 -16999.282,E2 -16999.282} C_VEL
LIN {X 0,Y 282.873,Z 768.465,A -85,B 0,C 180,E1 -17001.428,E2 -17001.428} C_VEL
LIN {X 0,Y 282.683,Z 770.179,A -85,B 0,C 180,E1 -17002.861,E2 -17002.861} C_VEL
LIN {X 0,Y 282.564,Z 771.436,A -85,B 0,C 180,E1 -17004.292,E2 -17004.292} C_VEL
LIN {X 0,Y 282.559,Z 772.291,A -85,B 0,C 180,E1 -17005.722,E2 -17005.722} C_VEL
LIN {X 0,Y 282.585,Z 772.748,A -85,B 0,C 180,E1 -17007.15,E2 -17007.15} C_VEL
LIN {X 0,Y 282.702,Z 772.79,A -85,B 0,C 180,E1 -17008.577,E2 -17008.577} C_VEL
LIN {X 0,Y 282.946,Z 772.379,A -85,B 0,C 180,E1 -17010.001,E2 -17010.001} C_VEL
LIN {X 0,Y 282.836,Z 771.523,A -85,B 0,C 180,E1 -17011.425,E2 -17011.425} C_VEL
LIN {X 0,Y 282.672,Z 770.24,A -85,B 0,C 180,E1 -17012.852,E2 -17012.852} C_VEL
LIN {X 0,Y 282.75,Z 767.444,A -85,B 0,C 180,E1 -17014.992,E2 -17014.992} C_VEL
LIN {X 0,Y 282.771,Z 763.525,A -85,B 0,C 180,E1 -17017.14,E2 -17017.14} C_VEL
LIN {X 0,Y 283.064,Z 757.374,A -85,B 0,C 180,E1 -17019.649,E2 -17019.649} C_VEL
LIN {X 0,Y 283.6,Z 750.626,A -85,B 0,C 180,E1 -17021.798,E2 -17021.798} C_VEL
LIN {X 0,Y 284.318,Z 743.735,A -85,B 0,C 180,E1 -17023.583,E2 -17023.583} C_VEL
LIN {X 0,Y 285.289,Z 735.451,A -85,B 0,C 180,E1 -17025.358,E2 -17025.358} C_VEL
LIN {X 0,Y 286.217,Z 726.932,A -85,B 0,C 180,E1 -17026.866,E2 -17026.866} C_VEL
LIN {X 0,Y 287.605,Z 715.367,A -85,B 0,C 180,E1 -17028.523,E2 -17028.523} C_VEL
LIN {X 0,Y 288.151,Z 707.946,A -85,B 0,C 180,E1 -17029.41,E2 -17029.41} C_VEL
LIN {X 0,Y 287.906,Z 694.774,A -85,B 0,C 180,E1 -17030.731,E2 -17030.731} C_VEL
LIN {X 0,Y 287.289,Z 681.312,A -85,B 0,C 180,E1 -17031.757,E2 -17031.757} C_VEL
LIN {X 0,Y 285.226,Z 657.135,A -85,B 0,C 180,E1 -17033.316,E2 -17033.316} C_VEL
LIN {X 0,Y 284.575,Z 651.471,A -85,B 0,C 180,E1 -17033.65,E2 -17033.65} C_VEL
LIN {X 0,Y 284.197,Z 643.297,A -85,B 0,C 180,E1 -17034.639,E2 -17034.639} C_VEL
LIN {X 0,Y 285.231,Z 633.313,A -85,B 0,C 180,E1 -17038.718,E2 -17038.718} C_VEL
LIN {X 0,Y 286.704,Z 621.589,A -85,B 0,C 180,E1 -17043.545,E2 -17043.545} C_VEL
LIN {X 0,Y 288.159,Z 611.961,A -85,B 0,C 180,E1 -17047.571,E2 -17047.571} C_VEL
LIN {X 0,Y 287.938,Z 607.841,A -85,B 0,C 180,E1 -17049.392,E2 -17049.392} C_VEL
LIN {X 0,Y 286.331,Z 599.342,A -85,B 0,C 180,E1 -17053.415,E2 -17053.415} C_VEL
LIN {X 0,Y 284.625,Z 590.63,A -85,B 0,C 180,E1 -17057.798,E2 -17057.798} C_VEL
LIN {X 0,Y 284.297,Z 589.074,A -85,B 0,C 180,E1 -17058.72,E2 -17058.72} C_VEL
LIN {X 0,Y 284.341,Z 589.072,A -85,B 0,C 180,E1 -17062.275,E2 -17062.275} C_VEL
LIN {X 0,Y 284.329,Z 589.069,A -85,B 0,C 180,E1 -17065.353,E2 -17065.353} C_VEL
LIN {X 0,Y 284.302,Z 589.072,A -85,B 0,C 180,E1 -17068.726,E2 -17068.726} C_VEL
LIN {X 0,Y 284.401,Z 589.057,A -85,B 0,C 180,E1 -17072.827,E2 -17072.827} C_VEL
LIN {X 0,Y 284.374,Z 589.062,A -85,B 0,C 180,E1 -17076.707,E2 -17076.707} C_VEL
LIN {X 0,Y 284.409,Z 589.056,A -85,B 0,C 180,E1 -17081.261,E2 -17081.261} C_VEL
LIN {X 0,Y 284.498,Z 589.05,A -85,B 0,C 180,E1 -17084.459,E2 -17084.459} C_VEL
LIN {X 0,Y 284.494,Z 589.048,A -85,B 0,C 180,E1 -17088.601,E2 -17088.601} C_VEL
LIN {X 0,Y 284.666,Z 589.023,A -85,B 0,C 180,E1 -17091.481,E2 -17091.481} C_VEL
